LIN {X 0,Y 177.073,Z 822.923,A -85,B 0,C 180,E1 -26070.539,E2 -26070.539} C_VEL
LIN {X 0,Y 180.629,Z 808.52,A -85,B 0,C 180,E1 -26071.33,E2 -26071.33} C_VEL
LIN {X 0,Y 182.9,Z 794.433,A -85,B 0,C 180,E1 -26071.841,E2 -26071.841} C_VEL
LIN {X 0,Y 185.471,Z 767.507,A -85,B 0,C 180,E1 -26072.606,E2 -26072.606} C_VEL
LIN {X 0,Y 182.681,Z 759.244,A -85,B 0,C 180,E1 -26075.344,E2 -26075.344} C_VEL
LIN {X 0,Y 179.682,Z 751.238,A -85,B 0,C 180,E1 -26078.707,E2 -26078.707} C_VEL
LIN {X 0,Y 177.784,Z 746.896,A -85,B 0,C 180,E1 -26081.141,E2 -26081.141} C_VEL
LIN {X 0,Y 176.059,Z 743.86,A -85,B 0,C 180,E1 -26083.611,E2 -26083.611} C_VEL
LIN {X 0,Y 174.842,Z 741.596,A -85,B 0,C 180,E1 -26085.711,E2 -26085.711} C_VEL
LIN {X 0,Y 172.904,Z 737.776,A -85,B 0,C 180,E1 -26090.311,E2 -26090.311} C_VEL
LIN {X 0,Y 171.638,Z 736.041,A -85,B 0,C 180,E1 -26097.654,E2 -26097.654} C_VEL
LIN {X 0,Y 171.809,Z 736.329,A -85,B 0,C 180,E1 -26100.587,E2 -26100.587} C_VEL
LIN {X 0,Y 173.048,Z 737.983,A -85,B 0,C 180,E1 -26105.682,E2 -26105.682} C_VEL
LIN {X 0,Y 174.768,Z 741.458,A -85,B 0,C 180,E1 -26109.725,E2 -26109.725} C_VEL
LIN {X 0,Y 175.622,Z 743.043,A -85,B 0,C 180,E1 -26111.251,E2 -26111.251} C_VEL
LIN {X 0,Y 177.589,Z 746.529,A -85,B 0,C 180,E1 -26114.175,E2 -26114.175} C_VEL
LIN {X 0,Y 180.001,Z 750.965,A -85,B 0,C 180,E1 -26117.129,E2 -26117.129} C_VEL
LIN {X 0,Y 183.401,Z 757.678,A -85,B 0,C 180,E1 -26120.615,E2 -26120.615} C_VEL
LIN {X 0,Y 185.832,Z 763.005,A -85,B 0,C 180,E1 -26122.807,E2 -26122.807} C_VEL
LIN {X 0,Y 182.965,Z 792.297,A -85,B 0,C 180,E1 -26123.684,E2 -26123.684} C_VEL
LIN {X 0,Y 180.308,Z 806.858,A -85,B 0,C 180,E1 -26124.351,E2 -26124.351} C_VEL
LIN {X 0,Y 176.455,Z 821.351,A -85,B 0,C 180,E1 -26125.363,E2 -26125.363} C_VEL
LIN {X 0,Y 171.502,Z 834.975,A -85,B 0,C 180,E1 -26126.6,E2 -26126.6} C_VEL
LIN {X 0,Y 166.318,Z 846.673,A -85,B 0,C 180,E1 -26128.103,E2 -26128.103} C_VEL
LIN {X 0,Y 160.284,Z 858.049,A -85,B 0,C 180,E1 -26130.005,E2 -26130.005} C_VEL
LIN {X 0,Y 153.748,Z 868.482,A -85,B 0,C 180,E1 -26132.258,E2 -26132.258} C_VEL
LIN {X 0,Y 146.256,Z 878.831,A -85,B 0,C 180,E1 -26135.225,E2 -26135.225} C_VEL
LIN {X 0,Y 139.276,Z 887.346,A -85,B 0,C 180,E1 -26138.543,E2 -26138.543} C_VEL
LIN {X 0,Y 131.602,Z 895.448,A -85,B 0,C 180,E1 -26142.752,E2 -26142.752} C_VEL
LIN {X 0,Y 124.73,Z 901.95,A -85,B 0,C 180,E1 -26147.457,E2 -26147.457} C_VEL
LIN {X 0,Y 117.992,Z 907.69,A -85,B 0,C 180,E1 -26153.443,E2 -26153.443} C_VEL
LIN {X 0,Y 112.636,Z 911.844,A -85,B 0,C 180,E1 -26160.055,E2 -26160.055} C_VEL
LIN {X 0,Y 108.658,Z 914.547,A -85,B 0,C 180,E1 -26167.165,E2 -26167.165} C_VEL
LIN {X 0,Y 106.159,Z 915.885,A -85,B 0,C 180,E1 -26174.645,E2 -26174.645} C_VEL
LIN {X 0,Y 105.229,Z 915.893,A -85,B 0,C 180,E1 -26182.324,E2 -26182.324} C_VEL
LIN {X 0,Y 105.422,Z 914.588,A -85,B 0,C 180,E1 -26190,E2 -26190} C_VEL
LIN {X 0,Y 106.561,Z 911.96,A -85,B 0,C 180,E1 -26197.58,E2 -26197.58} C_VEL
LIN {X 0,Y 109.233,Z 907.919,A -85,B 0,C 180,E1 -26204.914,E2 -26204.914} C_VEL
LIN {X 0,Y 112.051,Z 904.063,A -85,B 0,C 180,E1 -26209.989,E2 -26209.989} C_VEL
LIN {X 0,Y 115.769,Z 898.932,A -85,B 0,C 180,E1 -26215.148,E2 -26215.148} C_VEL
LIN {X 0,Y 120.816,Z 891.816,A -85,B 0,C 180,E1 -26220.597,E2 -26220.597} C_VEL
LIN {X 0,Y 127.127,Z 882.991,A -85,B 0,C 180,E1 -26225.485,E2 -26225.485} C_VEL
LIN {X 0,Y 133.06,Z 873.738,A -85,B 0,C 180,E1 -26229.333,E2 -26229.333} C_VEL
LIN {X 0,Y 138.745,Z 863.523,A -85,B 0,C 180,E1 -26232.649,E2 -26232.649} C_VEL
LIN {X 0,Y 142.557,Z 855.85,A -85,B 0,C 180,E1 -26234.63,E2 -26234.63} C_VEL
LIN {X 0,Y 147.858,Z 844.228,A -85,B 0,C 180,E1 -26236.954,E2 -26236.954} C_VEL
LIN {X 0,Y 152.056,Z 833.202,A -85,B 0,C 180,E1 -26238.684,E2 -26238.684} C_VEL
LIN {X 0,Y 156.398,Z 819.272,A -85,B 0,C 180,E1 -26240.313,E2 -26240.313} C_VEL
LIN {X 0,Y 159.627,Z 805.18,A -85,B 0,C 180,E1 -26241.524,E2 -26241.524} C_VEL
LIN {X 0,Y 161.82,Z 791.195,A -85,B 0,C 180,E1 -26242.321,E2 -26242.321} C_VEL
LIN {X 0,Y 165.759,Z 746.595,A -85,B 0,C 180,E1 -26243.808,E2 -26243.808} C_VEL
LIN {X 0,Y 161.599,Z 737.779,A -85,B 0,C 180,E1 -26246.875,E2 -26246.875} C_VEL
LIN {X 0,Y 157.468,Z 730.066,A -85,B 0,C 180,E1 -26250.312,E2 -26250.312} C_VEL
LIN {X 0,Y 153.944,Z 723.905,A -85,B 0,C 180,E1 -26253.732,E2 -26253.732} C_VEL
LIN {X 0,Y 151.674,Z 720.327,A -85,B 0,C 180,E1 -26256.257,E2 -26256.257} C_VEL
LIN {X 0,Y 149.381,Z 716.691,A -85,B 0,C 180,E1 -26259.241,E2 -26259.241} C_VEL
LIN {X 0,Y 147.032,Z 713.071,A -85,B 0,C 180,E1 -26263.011,E2 -26263.011} C_VEL
LIN {X 0,Y 144.407,Z 709.358,A -85,B 0,C 180,E1 -26269.192,E2 -26269.192} C_VEL
LIN {X 0,Y 143.974,Z 707.729,A -85,B 0,C 180,E1 -26271.246,E2 -26271.246} C_VEL
LIN {X 0,Y 143.41,Z 707.23,A -85,B 0,C 180,E1 -26279.999,E2 -26279.999} C_VEL
LIN {X 0,Y 144.182,Z 707.95,A -85,B 0,C 180,E1 -26284.105,E2 -26284.105} C_VEL
LIN {X 0,Y 145.926,Z 711.714,A -85,B 0,C 180,E1 -26289.355,E2 -26289.355} C_VEL
LIN {X 0,Y 147.111,Z 713.082,A -85,B 0,C 180,E1 -26291.617,E2 -26291.617} C_VEL
LIN {X 0,Y 149.448,Z 716.686,A -85,B 0,C 180,E1 -26295.338,E2 -26295.338} C_VEL
LIN {X 0,Y 152.699,Z 721.894,A -85,B 0,C 180,E1 -26299.414,E2 -26299.414} C_VEL
LIN {X 0,Y 156.291,Z 727.806,A -85,B 0,C 180,E1 -26303.082,E2 -26303.082} C_VEL
LIN {X 0,Y 158.506,Z 732.054,A -85,B 0,C 180,E1 -26305.103,E2 -26305.103} C_VEL
LIN {X 0,Y 161.92,Z 740.882,A -85,B 0,C 180,E1 -26308.077,E2 -26308.077} C_VEL
LIN {X 0,Y 165.49,Z 751.393,A -85,B 0,C 180,E1 -26310.914,E2 -26310.914} C_VEL
LIN {X 0,Y 161.322,Z 798.641,A -85,B 0,C 180,E1 -26312.498,E2 -26312.498} C_VEL
LIN {X 0,Y 158.933,Z 812.957,A -85,B 0,C 180,E1 -26313.276,E2 -26313.276} C_VEL
LIN {X 0,Y 155.415,Z 827.05,A -85,B 0,C 180,E1 -26314.382,E2 -26314.382} C_VEL
LIN {X 0,Y 150.891,Z 841.025,A -85,B 0,C 180,E1 -26315.975,E2 -26315.975} C_VEL
LIN {X 0,Y 145.821,Z 853.521,A -85,B 0,C 180,E1 -26317.888,E2 -26317.888} C_VEL
LIN {X 0,Y 140.409,Z 864.953,A -85,B 0,C 180,E1 -26320.241,E2 -26320.241} C_VEL
LIN {X 0,Y 134.823,Z 875.474,A -85,B 0,C 180,E1 -26323.131,E2 -26323.131} C_VEL
LIN {X 0,Y 128.441,Z 885.919,A -85,B 0,C 180,E1 -26326.844,E2 -26326.844} C_VEL
LIN {X 0,Y 122.678,Z 894.538,A -85,B 0,C 180,E1 -26330.937,E2 -26330.937} C_VEL
LIN {X 0,Y 116.942,Z 902.78,A -85,B 0,C 180,E1 -26336.226,E2 -26336.226} C_VEL
LIN {X 0,Y 112.117,Z 909.461,A -85,B 0,C 180,E1 -26342.013,E2 -26342.013} C_VEL
LIN {X 0,Y 108.319,Z 915.314,A -85,B 0,C 180,E1 -26349.092,E2 -26349.092} C_VEL
LIN {X 0,Y 106.388,Z 918.704,A -85,B 0,C 180,E1 -26354.678,E2 -26354.678} C_VEL
LIN {X 0,Y 105.229,Z 921.879,A -85,B 0,C 180,E1 -26362.323,E2 -26362.323} C_VEL
LIN {X 0,Y 105.149,Z 922.938,A -85,B 0,C 180,E1 -26366.167,E2 -26366.167} C_VEL
LIN {X 0,Y 105.301,Z 923.651,A -85,B 0,C 180,E1 -26370,E2 -26370} C_VEL
LIN {X 0,Y 105.224,Z 924.013,A -85,B 0,C 180,E1 -26377.676,E2 -26377.676} C_VEL
LIN {X 0,Y 106.436,Z 923.042,A -85,B 0,C 180,E1 -26385.314,E2 -26385.314} C_VEL
LIN {X 0,Y 109.333,Z 920.744,A -85,B 0,C 180,E1 -26392.686,E2 -26392.686} C_VEL
LIN {X 0,Y 113.857,Z 917.06,A -85,B 0,C 180,E1 -26399.591,E2 -26399.591} C_VEL
LIN {X 0,Y 119.273,Z 912.338,A -85,B 0,C 180,E1 -26405.452,E2 -26405.452} C_VEL
LIN {X 0,Y 121.304,Z 910.059,A -85,B 0,C 180,E1 -26407.862,E2 -26407.862} C_VEL
LIN {X 0,Y 123.493,Z 906.012,A -85,B 0,C 180,E1 -26411.974,E2 -26411.974} C_VEL
LIN {X 0,Y 126.146,Z 901.426,A -85,B 0,C 180,E1 -26415.814,E2 -26415.814} C_VEL
LIN {X 0,Y 128.79,Z 898.306,A -85,B 0,C 180,E1 -26417.725,E2 -26417.725} C_VEL
LIN {X 0,Y 136.909,Z 889.585,A -85,B 0,C 180,E1 -26421.521,E2 -26421.521} C_VEL
LIN {X 0,Y 144.395,Z 880.343,A -85,B 0,C 180,E1 -26424.492,E2 -26424.492} C_VEL
LIN {X 0,Y 151.862,Z 869.757,A -85,B 0,C 180,E1 -26427.014,E2 -26427.014} C_VEL
LIN {X 0,Y 158.865,Z 858.295,A -85,B 0,C 180,E1 -26428.995,E2 -26428.995} C_VEL
LIN {X 0,Y 164.572,Z 847.189,A -85,B 0,C 180,E1 -26430.471,E2 -26430.471} C_VEL
LIN {X 0,Y 169.642,Z 835.263,A -85,B 0,C 180,E1 -26431.685,E2 -26431.685} C_VEL
LIN {X 0,Y 174.075,Z 822.227,A -85,B 0,C 180,E1 -26432.65,E2 -26432.65} C_VEL
LIN {X 0,Y 177.7,Z 807.753,A -85,B 0,C 180,E1 -26433.406,E2 -26433.406} C_VEL
LIN {X 0,Y 179.983,Z 793.525,A -85,B 0,C 180,E1 -26433.91,E2 -26433.91} C_VEL
LIN {X 0,Y 182.27,Z 770.597,A -85,B 0,C 180,E1 -26434.526,E2 -26434.526} C_VEL
LIN {X 0,Y 179.677,Z 762.653,A -85,B 0,C 180,E1 -26437.393,E2 -26437.393} C_VEL
LIN {X 0,Y 177.483,Z 756.512,A -85,B 0,C 180,E1 -26440.166,E2 -26440.166} C_VEL
LIN {X 0,Y 176.003,Z 752.899,A -85,B 0,C 180,E1 -26442.274,E2 -26442.274} C_VEL
LIN {X 0,Y 173.64,Z 748.379,A -85,B 0,C 180,E1 -26446.261,E2 -26446.261} C_VEL
LIN {X 0,Y 171.931,Z 744.757,A -85,B 0,C 180,E1 -26450.59,E2 -26450.59} C_VEL
LIN {X 0,Y 170.77,Z 743.1,A -85,B 0,C 180,E1 -26457.642,E2 -26457.642} C_VEL
LIN {X 0,Y 170.939,Z 743.403,A -85,B 0,C 180,E1 -26460.59,E2 -26460.59} C_VEL
LIN {X 0,Y 171.974,Z 744.847,A -85,B 0,C 180,E1 -26465.13,E2 -26465.13} C_VEL
LIN {X 0,Y 173.727,Z 748.455,A -85,B 0,C 180,E1 -26469.47,E2 -26469.47} C_VEL
LIN {X 0,Y 176.152,Z 753.196,A -85,B 0,C 180,E1 -26473.52,E2 -26473.52} C_VEL
LIN {X 0,Y 178.871,Z 758.486,A -85,B 0,C 180,E1 -26476.992,E2 -26476.992} C_VEL
LIN {X 0,Y 182.507,Z 766.355,A -85,B 0,C 180,E1 -26480.809,E2 -26480.809} C_VEL
LIN {X 0,Y 182.607,Z 766.645,A -85,B 0,C 180,E1 -26480.911,E2 -26480.911} C_VEL
LIN {X 0,Y 179.863,Z 793.134,A -85,B 0,C 180,E1 -26481.688,E2 -26481.688} C_VEL
LIN {X 0,Y 177.112,Z 807.587,A -85,B 0,C 180,E1 -26482.34,E2 -26482.34} C_VEL
LIN {X 0,Y 173.154,Z 821.94,A -85,B 0,C 180,E1 -26483.321,E2 -26483.321} C_VEL
LIN {X 0,Y 168.297,Z 834.919,A -85,B 0,C 180,E1 -26484.459,E2 -26484.459} C_VEL
LIN {X 0,Y 163.066,Z 846.428,A -85,B 0,C 180,E1 -26485.882,E2 -26485.882} C_VEL
LIN {X 0,Y 156.137,Z 859.073,A -85,B 0,C 180,E1 -26487.95,E2 -26487.95} C_VEL
LIN {X 0,Y 150.035,Z 868.401,A -85,B 0,C 180,E1 -26489.936,E2 -26489.936} C_VEL
LIN {X 0,Y 142.248,Z 878.818,A -85,B 0,C 180,E1 -26492.869,E2 -26492.869} C_VEL
LIN {X 0,Y 134.919,Z 887.383,A -85,B 0,C 180,E1 -26496.158,E2 -26496.158} C_VEL
LIN {X 0,Y 126.828,Z 895.54,A -85,B 0,C 180,E1 -26500.365,E2 -26500.365} C_VEL
LIN {X 0,Y 119.532,Z 902.079,A -85,B 0,C 180,E1 -26505.126,E2 -26505.126} C_VEL
LIN {X 0,Y 112.286,Z 907.853,A -85,B 0,C 180,E1 -26511.252,E2 -26511.252} C_VEL
LIN {X 0,Y 106.461,Z 912.039,A -85,B 0,C 180,E1 -26518.122,E2 -26518.122} C_VEL
LIN {X 0,Y 102.067,Z 914.772,A -85,B 0,C 180,E1 -26525.598,E2 -26525.598} C_VEL
LIN {X 0,Y 99.251,Z 916.139,A -85,B 0,C 180,E1 -26533.547,E2 -26533.547} C_VEL
LIN {X 0,Y 98.161,Z 916.177,A -85,B 0,C 180,E1 -26541.768,E2 -26541.768} C_VEL
LIN {X 0,Y 98.316,Z 914.907,A -85,B 0,C 180,E1 -26550,E2 -26550} C_VEL
LIN {X 0,Y 99.549,Z 912.313,A -85,B 0,C 180,E1 -26558.118,E2 -26558.118} C_VEL
LIN {X 0,Y 102.417,Z 908.303,A -85,B 0,C 180,E1 -26565.932,E2 -26565.932} C_VEL
LIN {X 0,Y 105.534,Z 904.324,A -85,B 0,C 180,E1 -26571.486,E2 -26571.486} C_VEL
LIN {X 0,Y 109.397,Z 899.368,A -85,B 0,C 180,E1 -26576.725,E2 -26576.725} C_VEL
LIN {X 0,Y 114.789,Z 892.289,A -85,B 0,C 180,E1 -26582.393,E2 -26582.393} C_VEL
LIN {X 0,Y 121.449,Z 883.509,A -85,B 0,C 180,E1 -26587.418,E2 -26587.418} C_VEL
LIN {X 0,Y 127.682,Z 874.314,A -85,B 0,C 180,E1 -26591.34,E2 -26591.34} C_VEL
LIN {X 0,Y 133.645,Z 864.172,A -85,B 0,C 180,E1 -26594.697,E2 -26594.697} C_VEL
LIN {X 0,Y 137.63,Z 856.543,A -85,B 0,C 180,E1 -26596.692,E2 -26596.692} C_VEL
LIN {X 0,Y 143.12,Z 845.016,A -85,B 0,C 180,E1 -26599.026,E2 -26599.026} C_VEL
LIN {X 0,Y 148.149,Z 832.352,A -85,B 0,C 180,E1 -26600.97,E2 -26600.97} C_VEL
LIN {X 0,Y 152.321,Z 819.233,A -85,B 0,C 180,E1 -26602.469,E2 -26602.469} C_VEL
LIN {X 0,Y 155.676,Z 805.031,A -85,B 0,C 180,E1 -26603.665,E2 -26603.665} C_VEL
LIN {X 0,Y 157.936,Z 790.7,A -85,B 0,C 180,E1 -26604.46,E2 -26604.46} C_VEL
LIN {X 0,Y 161.683,Z 750.383,A -85,B 0,C 180,E1 -26605.753,E2 -26605.753} C_VEL
LIN {X 0,Y 161.578,Z 749.318,A -85,B 0,C 180,E1 -26605.904,E2 -26605.904} C_VEL
LIN {X 0,Y 157.893,Z 741.409,A -85,B 0,C 180,E1 -26608.92,E2 -26608.92} C_VEL
LIN {X 0,Y 153.683,Z 733.209,A -85,B 0,C 180,E1 -26612.898,E2 -26612.898} C_VEL
LIN {X 0,Y 150.227,Z 727.144,A -85,B 0,C 180,E1 -26616.813,E2 -26616.813} C_VEL
LIN {X 0,Y 147.749,Z 723.204,A -85,B 0,C 180,E1 -26620.212,E2 -26620.212} C_VEL
LIN {X 0,Y 145.313,Z 719.255,A -85,B 0,C 180,E1 -26624.549,E2 -26624.549} C_VEL
LIN {X 0,Y 143.413,Z 716.402,A -85,B 0,C 180,E1 -26629.537,E2 -26629.537} C_VEL
LIN {X 0,Y 143.022,Z 714.868,A -85,B 0,C 180,E1 -26631.522,E2 -26631.522} C_VEL
LIN {X 0,Y 142.542,Z 714.285,A -85,B 0,C 180,E1 -26639.999,E2 -26639.999} C_VEL
LIN {X 0,Y 143.167,Z 714.938,A -85,B 0,C 180,E1 -26643.583,E2 -26643.583} C_VEL
LIN {X 0,Y 144.958,Z 718.789,A -85,B 0,C 180,E1 -26649.207,E2 -26649.207} C_VEL
LIN {X 0,Y 145.799,Z 719.875,A -85,B 0,C 180,E1 -26650.906,E2 -26650.906} C_VEL
LIN {X 0,Y 148.461,Z 724.292,A -85,B 0,C 180,E1 -26655.333,E2 -26655.333} C_VEL
LIN {X 0,Y 151.218,Z 728.929,A -85,B 0,C 180,E1 -26658.897,E2 -26658.897} C_VEL
LIN {X 0,Y 154.178,Z 734.124,A -85,B 0,C 180,E1 -26662.1,E2 -26662.1} C_VEL
LIN {X 0,Y 156.02,Z 737.94,A -85,B 0,C 180,E1 -26663.916,E2 -26663.916} C_VEL
LIN {X 0,Y 159.188,Z 746.807,A -85,B 0,C 180,E1 -26666.916,E2 -26666.916} C_VEL
LIN {X 0,Y 161.451,Z 753.905,A -85,B 0,C 180,E1 -26668.899,E2 -26668.899} C_VEL
LIN {X 0,Y 157.348,Z 798.562,A -85,B 0,C 180,E1 -26670.39,E2 -26670.39} C_VEL
LIN {X 0,Y 154.79,Z 813.184,A -85,B 0,C 180,E1 -26671.176,E2 -26671.176} C_VEL
LIN {X 0,Y 151.159,Z 827.148,A -85,B 0,C 180,E1 -26672.262,E2 -26672.262} C_VEL
LIN {X 0,Y 146.8,Z 840.151,A -85,B 0,C 180,E1 -26673.713,E2 -26673.713} C_VEL
LIN {X 0,Y 141.543,Z 852.763,A -85,B 0,C 180,E1 -26675.603,E2 -26675.603} C_VEL
LIN {X 0,Y 135.899,Z 864.281,A -85,B 0,C 180,E1 -26677.94,E2 -26677.94} C_VEL
LIN {X 0,Y 130.037,Z 874.868,A -85,B 0,C 180,E1 -26680.83,E2 -26680.83} C_VEL
LIN {X 0,Y 123.323,Z 885.374,A -85,B 0,C 180,E1 -26684.572,E2 -26684.572} C_VEL
LIN {X 0,Y 117.181,Z 894.037,A -85,B 0,C 180,E1 -26688.72,E2 -26688.72} C_VEL
LIN {X 0,Y 111.064,Z 902.336,A -85,B 0,C 180,E1 -26694.173,E2 -26694.173} C_VEL
LIN {X 0,Y 105.664,Z 909.265,A -85,B 0,C 180,E1 -26700.426,E2 -26700.426} C_VEL
LIN {X 0,Y 101.675,Z 914.936,A -85,B 0,C 180,E1 -26707.655,E2 -26707.655} C_VEL
LIN {X 0,Y 99.504,Z 918.354,A -85,B 0,C 180,E1 -26713.589,E2 -26713.589} C_VEL
LIN {X 0,Y 98.171,Z 921.558,A -85,B 0,C 180,E1 -26721.768,E2 -26721.768} C_VEL
LIN {X 0,Y 98.066,Z 922.632,A -85,B 0,C 180,E1 -26725.89,E2 -26725.89} C_VEL
LIN {X 0,Y 98.2,Z 923.358,A -85,B 0,C 180,E1 -26730,E2 -26730} C_VEL
LIN {X 0,Y 98.167,Z 923.745,A -85,B 0,C 180,E1 -26738.232,E2 -26738.232} C_VEL
LIN {X 0,Y 99.572,Z 922.801,A -85,B 0,C 180,E1 -26746.399,E2 -26746.399} C_VEL
LIN {X 0,Y 102.778,Z 920.529,A -85,B 0,C 180,E1 -26754.222,E2 -26754.222} C_VEL
LIN {X 0,Y 107.673,Z 916.874,A -85,B 0,C 180,E1 -26761.478,E2 -26761.478} C_VEL
LIN {X 0,Y 114.069,Z 911.733,A -85,B 0,C 180,E1 -26768.033,E2 -26768.033} C_VEL
LIN {X 0,Y 119.82,Z 906.784,A -85,B 0,C 180,E1 -26772.417,E2 -26772.417} C_VEL
LIN {X 0,Y 127.356,Z 899.704,A -85,B 0,C 180,E1 -26776.986,E2 -26776.986} C_VEL
LIN {X 0,Y 128.79,Z 898.306,A -85,B 0,C 180,E1 -26777.725,E2 -26777.725} C_VEL
LIN {X 0,Y 131.53,Z 895.029,A -85,B 0,C 180,E1 -26779.529,E2 -26779.529} C_VEL
LIN {X 0,Y 134.869,Z 889.483,A -85,B 0,C 180,E1 -26782.77,E2 -26782.77} C_VEL
LIN {X 0,Y 138.31,Z 883.455,A -85,B 0,C 180,E1 -26785.745,E2 -26785.745} C_VEL
LIN {X 0,Y 141.092,Z 879.427,A -85,B 0,C 180,E1 -26787.104,E2 -26787.104} C_VEL
LIN {X 0,Y 148.829,Z 868.775,A -85,B 0,C 180,E1 -26789.519,E2 -26789.519} C_VEL
LIN {X 0,Y 156.04,Z 857.167,A -85,B 0,C 180,E1 -26791.435,E2 -26791.435} C_VEL
LIN {X 0,Y 162.684,Z 844.289,A -85,B 0,C 180,E1 -26793,E2 -26793} C_VEL
LIN {X 0,Y 168.302,Z 830.696,A -85,B 0,C 180,E1 -26794.212,E2 -26794.212} C_VEL
LIN {X 0,Y 172.636,Z 817.104,A -85,B 0,C 180,E1 -26795.067,E2 -26795.067} C_VEL
LIN {X 0,Y 175.903,Z 802.401,A -85,B 0,C 180,E1 -26795.724,E2 -26795.724} C_VEL
LIN {X 0,Y 177.927,Z 787.042,A -85,B 0,C 180,E1 -26796.179,E2 -26796.179} C_VEL
LIN {X 0,Y 179.248,Z 773.696,A -85,B 0,C 180,E1 -26796.538,E2 -26796.538} C_VEL
LIN {X 0,Y 176.676,Z 765.423,A -85,B 0,C 180,E1 -26799.821,E2 -26799.821} C_VEL
LIN {X 0,Y 174.789,Z 760.013,A -85,B 0,C 180,E1 -26802.638,E2 -26802.638} C_VEL
LIN {X 0,Y 172.66,Z 755.489,A -85,B 0,C 180,E1 -26806.405,E2 -26806.405} C_VEL
LIN {X 0,Y 170.88,Z 751.655,A -85,B 0,C 180,E1 -26811.128,E2 -26811.128} C_VEL
LIN {X 0,Y 169.903,Z 750.158,A -85,B 0,C 180,E1 -26817.63,E2 -26817.63} C_VEL
LIN {X 0,Y 170.103,Z 750.573,A -85,B 0,C 180,E1 -26820.888,E2 -26820.888} C_VEL
LIN {X 0,Y 170.992,Z 751.965,A -85,B 0,C 180,E1 -26824.864,E2 -26824.864} C_VEL
LIN {X 0,Y 172.819,Z 755.943,A -85,B 0,C 180,E1 -26829.52,E2 -26829.52} C_VEL
LIN {X 0,Y 174.701,Z 759.82,A -85,B 0,C 180,E1 -26832.802,E2 -26832.802} C_VEL
LIN {X 0,Y 177.124,Z 764.87,A -85,B 0,C 180,E1 -26836.127,E2 -26836.127} C_VEL
LIN {X 0,Y 179.522,Z 770.357,A -85,B 0,C 180,E1 -26838.902,E2 -26838.902} C_VEL
LIN {X 0,Y 177.057,Z 793.466,A -85,B 0,C 180,E1 -26839.598,E2 -26839.598} C_VEL
LIN {X 0,Y 174.237,Z 807.881,A -85,B 0,C 180,E1 -26840.225,E2 -26840.225} C_VEL
LIN {X 0,Y 170.45,Z 821.39,A -85,B 0,C 180,E1 -26841.113,E2 -26841.113} C_VEL
LIN {X 0,Y 165.339,Z 834.849,A -85,B 0,C 180,E1 -26842.233,E2 -26842.233} C_VEL
LIN {X 0,Y 160.067,Z 846.182,A -85,B 0,C 180,E1 -26843.574,E2 -26843.574} C_VEL
LIN {X 0,Y 153.615,Z 857.742,A -85,B 0,C 180,E1 -26845.368,E2 -26845.368} C_VEL
LIN {X 0,Y 146.585,Z 868.32,A -85,B 0,C 180,E1 -26847.504,E2 -26847.504} C_VEL
LIN {X 0,Y 138.484,Z 878.798,A -85,B 0,C 180,E1 -26850.374,E2 -26850.374} C_VEL
LIN {X 0,Y 130.81,Z 887.413,A -85,B 0,C 180,E1 -26853.617,E2 -26853.617} C_VEL
LIN {X 0,Y 122.3,Z 895.633,A -85,B 0,C 180,E1 -26857.801,E2 -26857.801} C_VEL
LIN {X 0,Y 114.546,Z 902.208,A -85,B 0,C 180,E1 -26862.586,E2 -26862.586} C_VEL
LIN {X 0,Y 106.76,Z 908.016,A -85,B 0,C 180,E1 -26868.83,E2 -26868.83} C_VEL
LIN {X 0,Y 100.404,Z 912.235,A -85,B 0,C 180,E1 -26875.946,E2 -26875.946} C_VEL
LIN {X 0,Y 95.565,Z 914.998,A -85,B 0,C 180,E1 -26883.817,E2 -26883.817} C_VEL
LIN {X 0,Y 92.389,Z 916.393,A -85,B 0,C 180,E1 -26892.286,E2 -26892.286} C_VEL
LIN {X 0,Y 91.101,Z 916.458,A -85,B 0,C 180,E1 -26901.125,E2 -26901.125} C_VEL
LIN {X 0,Y 91.219,Z 915.221,A -85,B 0,C 180,E1 -26910,E2 -26910} C_VEL
LIN {X 0,Y 92.549,Z 912.664,A -85,B 0,C 180,E1 -26918.736,E2 -26918.736} C_VEL
LIN {X 0,Y 95.632,Z 908.687,A -85,B 0,C 180,E1 -26927.096,E2 -26927.096} C_VEL
LIN {X 0,Y 98.977,Z 904.725,A -85,B 0,C 180,E1 -26932.988,E2 -26932.988} C_VEL
LIN {X 0,Y 103.132,Z 899.803,A -85,B 0,C 180,E1 -26938.491,E2 -26938.491} C_VEL
LIN {X 0,Y 108.891,Z 892.761,A -85,B 0,C 180,E1 -26944.385,E2 -26944.385} C_VEL
LIN {X 0,Y 115.923,Z 884.023,A -85,B 0,C 180,E1 -26949.538,E2 -26949.538} C_VEL
LIN {X 0,Y 122.476,Z 874.88,A -85,B 0,C 180,E1 -26953.519,E2 -26953.519} C_VEL
LIN {X 0,Y 128.731,Z 864.807,A -85,B 0,C 180,E1 -26956.904,E2 -26956.904} C_VEL
LIN {X 0,Y 132.895,Z 857.235,A -85,B 0,C 180,E1 -26958.903,E2 -26958.903} C_VEL
LIN {X 0,Y 138.589,Z 845.801,A -85,B 0,C 180,E1 -26961.232,E2 -26961.232} C_VEL
LIN {X 0,Y 143.816,Z 833.258,A -85,B 0,C 180,E1 -26963.151,E2 -26963.151} C_VEL
LIN {X 0,Y 148.138,Z 820.316,A -85,B 0,C 180,E1 -26964.629,E2 -26964.629} C_VEL
LIN {X 0,Y 151.613,Z 806.399,A -85,B 0,C 180,E1 -26965.807,E2 -26965.807} C_VEL
LIN {X 0,Y 154.074,Z 792.037,A -85,B 0,C 180,E1 -26966.617,E2 -26966.617} C_VEL
LIN {X 0,Y 157.813,Z 752.619,A -85,B 0,C 180,E1 -26967.932,E2 -26967.932} C_VEL
LIN {X 0,Y 154.16,Z 744.623,A -85,B 0,C 180,E1 -26971.285,E2 -26971.285} C_VEL
LIN {X 0,Y 150.312,Z 736.877,A -85,B 0,C 180,E1 -26975.458,E2 -26975.458} C_VEL
LIN {X 0,Y 147.838,Z 732.613,A -85,B 0,C 180,E1 -26978.637,E2 -26978.637} C_VEL
LIN {X 0,Y 146.181,Z 729.715,A -85,B 0,C 180,E1 -26981.176,E2 -26981.176} C_VEL
LIN {X 0,Y 144.101,Z 726.071,A -85,B 0,C 180,E1 -26985.191,E2 -26985.191} C_VEL
LIN {X 0,Y 142.332,Z 723.152,A -85,B 0,C 180,E1 -26990.303,E2 -26990.303} C_VEL
LIN {X 0,Y 142.03,Z 721.788,A -85,B 0,C 180,E1 -26992.106,E2 -26992.106} C_VEL
LIN {X 0,Y 141.678,Z 721.311,A -85,B 0,C 180,E1 -26999.999,E2 -26999.999} C_VEL
LIN {X 0,Y 142.17,Z 721.881,A -85,B 0,C 180,E1 -27003.054,E2 -27003.054} C_VEL
LIN {X 0,Y 143.805,Z 725.652,A -85,B 0,C 180,E1 -27008.643,E2 -27008.643} C_VEL
LIN {X 0,Y 144.592,Z 726.849,A -85,B 0,C 180,E1 -27010.364,E2 -27010.364} C_VEL
LIN {X 0,Y 146.858,Z 730.79,A -85,B 0,C 180,E1 -27014.395,E2 -27014.395} C_VEL
LIN {X 0,Y 149.399,Z 735.345,A -85,B 0,C 180,E1 -27017.937,E2 -27017.937} C_VEL
LIN {X 0,Y 152.045,Z 740.252,A -85,B 0,C 180,E1 -27021.013,E2 -27021.013} C_VEL
LIN {X 0,Y 153.558,Z 743.659,A -85,B 0,C 180,E1 -27022.638,E2 -27022.638} C_VEL
LIN {X 0,Y 156.452,Z 752.491,A -85,B 0,C 180,E1 -27025.644,E2 -27025.644} C_VEL
LIN {X 0,Y 157.605,Z 756.445,A -85,B 0,C 180,E1 -27026.775,E2 -27026.775} C_VEL
LIN {X 0,Y 153.57,Z 798.621,A -85,B 0,C 180,E1 -27028.178,E2 -27028.178} C_VEL
LIN {X 0,Y 151.047,Z 812.646,A -85,B 0,C 180,E1 -27028.917,E2 -27028.917} C_VEL
LIN {X 0,Y 147.47,Z 826.108,A -85,B 0,C 180,E1 -27029.914,E2 -27029.914} C_VEL
LIN {X 0,Y 142.958,Z 839.278,A -85,B 0,C 180,E1 -27031.33,E2 -27031.33} C_VEL
LIN {X 0,Y 137.52,Z 852.008,A -85,B 0,C 180,E1 -27033.19,E2 -27033.19} C_VEL
LIN {X 0,Y 131.608,Z 863.606,A -85,B 0,C 180,E1 -27035.475,E2 -27035.475} C_VEL
LIN {X 0,Y 125.468,Z 874.262,A -85,B 0,C 180,E1 -27038.353,E2 -27038.353} C_VEL
LIN {X 0,Y 118.418,Z 884.824,A -85,B 0,C 180,E1 -27042.109,E2 -27042.109} C_VEL
LIN {X 0,Y 111.883,Z 893.531,A -85,B 0,C 180,E1 -27046.292,E2 -27046.292} C_VEL
LIN {X 0,Y 105.353,Z 901.89,A -85,B 0,C 180,E1 -27051.898,E2 -27051.898} C_VEL
LIN {X 0,Y 99.7,Z 908.543,A -85,B 0,C 180,E1 -27058.018,E2 -27058.018} C_VEL
LIN {X 0,Y 96.082,Z 913.232,A -85,B 0,C 180,E1 -27063.967,E2 -27063.967} C_VEL
LIN {X 0,Y 92.666,Z 917.998,A -85,B 0,C 180,E1 -27072.34,E2 -27072.34} C_VEL
LIN {X 0,Y 91.119,Z 921.237,A -85,B 0,C 180,E1 -27081.126,E2 -27081.126} C_VEL
LIN {X 0,Y 90.98,Z 922.325,A -85,B 0,C 180,E1 -27085.569,E2 -27085.569} C_VEL
LIN {X 0,Y 91.111,Z 923.065,A -85,B 0,C 180,E1 -27090,E2 -27090} C_VEL
LIN {X 0,Y 91.117,Z 923.477,A -85,B 0,C 180,E1 -27098.874,E2 -27098.874} C_VEL
LIN {X 0,Y 92.736,Z 922.56,A -85,B 0,C 180,E1 -27107.646,E2 -27107.646} C_VEL
LIN {X 0,Y 96.312,Z 920.316,A -85,B 0,C 180,E1 -27115.965,E2 -27115.965} C_VEL
LIN {X 0,Y 101.625,Z 916.688,A -85,B 0,C 180,E1 -27123.59,E2 -27123.59} C_VEL
LIN {X 0,Y 108.52,Z 911.578,A -85,B 0,C 180,E1 -27130.362,E2 -27130.362} C_VEL
LIN {X 0,Y 116.8,Z 904.836,A -85,B 0,C 180,E1 -27136.224,E2 -27136.224} C_VEL
LIN {X 0,Y 125.043,Z 897.346,A -85,B 0,C 180,E1 -27140.607,E2 -27140.607} C_VEL
LIN {X 0,Y 133.798,Z 888.22,A -85,B 0,C 180,E1 -27144.379,E2 -27144.379} C_VEL
LIN {X 0,Y 141.092,Z 879.427,A -85,B 0,C 180,E1 -27147.104,E2 -27147.104} C_VEL
LIN {X 0,Y 143.885,Z 875.298,A -85,B 0,C 180,E1 -27148.378,E2 -27148.378} C_VEL
LIN {X 0,Y 147.364,Z 868.35,A -85,B 0,C 180,E1 -27150.806,E2 -27150.806} C_VEL
LIN {X 0,Y 150.809,Z 861.081,A -85,B 0,C 180,E1 -27153.007,E2 -27153.007} C_VEL
LIN {X 0,Y 153.374,Z 856.309,A -85,B 0,C 180,E1 -27153.904,E2 -27153.904} C_VEL
LIN {X 0,Y 159.597,Z 844.547,A -85,B 0,C 180,E1 -27155.263,E2 -27155.263} C_VEL
LIN {X 0,Y 164.958,Z 832.082,A -85,B 0,C 180,E1 -27156.348,E2 -27156.348} C_VEL
LIN {X 0,Y 169.29,Z 819.323,A -85,B 0,C 180,E1 -27157.15,E2 -27157.15} C_VEL
LIN {X 0,Y 172.819,Z 805.081,A -85,B 0,C 180,E1 -27157.796,E2 -27157.796} C_VEL
LIN {X 0,Y 174.985,Z 791.244,A -85,B 0,C 180,E1 -27158.218,E2 -27158.218} C_VEL
LIN {X 0,Y 176.429,Z 776.975,A -85,B 0,C 180,E1 -27158.619,E2 -27158.619} C_VEL
LIN {X 0,Y 174.164,Z 769.113,A -85,B 0,C 180,E1 -27162.005,E2 -27162.005} C_VEL
LIN {X 0,Y 172.861,Z 765.424,A -85,B 0,C 180,E1 -27164.234,E2 -27164.234} C_VEL
LIN {X 0,Y 171.138,Z 761.753,A -85,B 0,C 180,E1 -27167.701,E2 -27167.701} C_VEL
LIN {X 0,Y 169.896,Z 758.62,A -85,B 0,C 180,E1 -27171.49,E2 -27171.49} C_VEL
LIN {X 0,Y 169.036,Z 757.217,A -85,B 0,C 180,E1 -27177.618,E2 -27177.618} C_VEL
LIN {X 0,Y 169.23,Z 757.677,A -85,B 0,C 180,E1 -27180.893,E2 -27180.893} C_VEL
LIN {X 0,Y 169.98,Z 758.925,A -85,B 0,C 180,E1 -27184.447,E2 -27184.447} C_VEL
LIN {X 0,Y 171.643,Z 762.832,A -85,B 0,C 180,E1 -27189.009,E2 -27189.009} C_VEL
LIN {X 0,Y 173.323,Z 766.532,A -85,B 0,C 180,E1 -27192.143,E2 -27192.143} C_VEL
LIN {X 0,Y 175.535,Z 771.459,A -85,B 0,C 180,E1 -27195.392,E2 -27195.392} C_VEL
LIN {X 0,Y 176.671,Z 774.478,A -85,B 0,C 180,E1 -27196.881,E2 -27196.881} C_VEL
LIN {X 0,Y 174.358,Z 794.644,A -85,B 0,C 180,E1 -27197.477,E2 -27197.477} C_VEL
LIN {X 0,Y 171.347,Z 809.215,A -85,B 0,C 180,E1 -27198.095,E2 -27198.095} C_VEL
LIN {X 0,Y 167.245,Z 823.116,A -85,B 0,C 180,E1 -27199.004,E2 -27199.004} C_VEL
LIN {X 0,Y 162.638,Z 834.784,A -85,B 0,C 180,E1 -27199.932,E2 -27199.932} C_VEL
LIN {X 0,Y 157.337,Z 845.937,A -85,B 0,C 180,E1 -27201.18,E2 -27201.18} C_VEL
LIN {X 0,Y 150.689,Z 857.589,A -85,B 0,C 180,E1 -27202.909,E2 -27202.909} C_VEL
LIN {X 0,Y 143.41,Z 868.24,A -85,B 0,C 180,E1 -27204.959,E2 -27204.959} C_VEL
LIN {X 0,Y 134.992,Z 878.776,A -85,B 0,C 180,E1 -27207.741,E2 -27207.741} C_VEL
LIN {X 0,Y 126.963,Z 887.442,A -85,B 0,C 180,E1 -27210.908,E2 -27210.908} C_VEL
LIN {X 0,Y 118.037,Z 895.722,A -85,B 0,C 180,E1 -27215.047,E2 -27215.047} C_VEL
LIN {X 0,Y 109.826,Z 902.337,A -85,B 0,C 180,E1 -27219.834,E2 -27219.834} C_VEL
LIN {X 0,Y 101.445,Z 908.18,A -85,B 0,C 180,E1 -27226.149,E2 -27226.149} C_VEL
LIN {X 0,Y 94.522,Z 912.43,A -85,B 0,C 180,E1 -27233.5,E2 -27233.5} C_VEL
LIN {X 0,Y 89.169,Z 915.223,A -85,B 0,C 180,E1 -27241.778,E2 -27241.778} C_VEL
LIN {X 0,Y 85.583,Z 916.648,A -85,B 0,C 180,E1 -27250.824,E2 -27250.824} C_VEL
LIN {X 0,Y 84.042,Z 916.741,A -85,B 0,C 180,E1 -27260.372,E2 -27260.372} C_VEL
LIN {X 0,Y 83.902,Z 916.298,A -85,B 0,C 180,E1 -27265.195,E2 -27265.195} C_VEL
LIN {X 0,Y 84.67,Z 914.439,A -85,B 0,C 180,E1 -27274.762,E2 -27274.762} C_VEL
LIN {X 0,Y 86.979,Z 911.227,A -85,B 0,C 180,E1 -27284.029,E2 -27284.029} C_VEL
LIN {X 0,Y 91.286,Z 906.53,A -85,B 0,C 180,E1 -27292.641,E2 -27292.641} C_VEL
LIN {X 0,Y 96.963,Z 900.238,A -85,B 0,C 180,E1 -27300.489,E2 -27300.489} C_VEL
LIN {X 0,Y 103.142,Z 893.233,A -85,B 0,C 180,E1 -27306.6,E2 -27306.6} C_VEL
LIN {X 0,Y 110.572,Z 884.538,A -85,B 0,C 180,E1 -27311.866,E2 -27311.866} C_VEL
LIN {X 0,Y 117.464,Z 875.444,A -85,B 0,C 180,E1 -27315.888,E2 -27315.888} C_VEL
LIN {X 0,Y 124.653,Z 864.427,A -85,B 0,C 180,E1 -27319.565,E2 -27319.565} C_VEL
LIN {X 0,Y 130.956,Z 853.183,A -85,B 0,C 180,E1 -27322.335,E2 -27322.335} C_VEL
LIN {X 0,Y 136.968,Z 840.724,A -85,B 0,C 180,E1 -27324.545,E2 -27324.545} C_VEL
LIN {X 0,Y 141.773,Z 828.674,A -85,B 0,C 180,E1 -27326.134,E2 -27326.134} C_VEL
LIN {X 0,Y 145.883,Z 815.441,A -85,B 0,C 180,E1 -27327.467,E2 -27327.467} C_VEL
LIN {X 0,Y 149.123,Z 801.179,A -85,B 0,C 180,E1 -27328.483,E2 -27328.483} C_VEL
LIN {X 0,Y 151.186,Z 787.067,A -85,B 0,C 180,E1 -27329.127,E2 -27329.127} C_VEL
LIN {X 0,Y 154.148,Z 755.819,A -85,B 0,C 180,E1 -27330.145,E2 -27330.145} C_VEL
LIN {X 0,Y 150.74,Z 748.082,A -85,B 0,C 180,E1 -27333.701,E2 -27333.701} C_VEL
LIN {X 0,Y 147.767,Z 741.984,A -85,B 0,C 180,E1 -27337.357,E2 -27337.357} C_VEL
LIN {X 0,Y 145.076,Z 736.801,A -85,B 0,C 180,E1 -27341.451,E2 -27341.451} C_VEL
LIN {X 0,Y 142.938,Z 732.936,A -85,B 0,C 180,E1 -27345.768,E2 -27345.768} C_VEL
LIN {X 0,Y 141.279,Z 729.912,A -85,B 0,C 180,E1 -27351.069,E2 -27351.069} C_VEL
LIN {X 0,Y 141.02,Z 728.751,A -85,B 0,C 180,E1 -27352.841,E2 -27352.841} C_VEL
LIN {X 0,Y 140.897,Z 728.464,A -85,B 0,C 180,E1 -27360.741,E2 -27360.741} C_VEL
LIN {X 0,Y 141.208,Z 728.944,A -85,B 0,C 180,E1 -27362.68,E2 -27362.68} C_VEL
LIN {X 0,Y 142.77,Z 732.614,A -85,B 0,C 180,E1 -27368.313,E2 -27368.313} C_VEL
LIN {X 0,Y 143.613,Z 734.289,A -85,B 0,C 180,E1 -27370.292,E2 -27370.292} C_VEL
LIN {X 0,Y 145.422,Z 737.52,A -85,B 0,C 180,E1 -27373.648,E2 -27373.648} C_VEL
LIN {X 0,Y 147.841,Z 742.129,A -85,B 0,C 180,E1 -27377.239,E2 -27377.239} C_VEL
LIN {X 0,Y 150.616,Z 747.751,A -85,B 0,C 180,E1 -27380.644,E2 -27380.644} C_VEL
LIN {X 0,Y 153.043,Z 755.603,A -85,B 0,C 180,E1 -27383.502,E2 -27383.502} C_VEL
LIN {X 0,Y 153.99,Z 758.99,A -85,B 0,C 180,E1 -27384.551,E2 -27384.551} C_VEL
LIN {X 0,Y 150.26,Z 797.176,A -85,B 0,C 180,E1 -27385.797,E2 -27385.797} C_VEL
LIN {X 0,Y 147.718,Z 811.335,A -85,B 0,C 180,E1 -27386.485,E2 -27386.485} C_VEL
LIN {X 0,Y 144.046,Z 825.069,A -85,B 0,C 180,E1 -27387.455,E2 -27387.455} C_VEL
LIN {X 0,Y 139.397,Z 838.41,A -85,B 0,C 180,E1 -27388.836,E2 -27388.836} C_VEL
LIN {X 0,Y 133.758,Z 851.254,A -85,B 0,C 180,E1 -27390.639,E2 -27390.639} C_VEL
LIN {X 0,Y 127.58,Z 862.931,A -85,B 0,C 180,E1 -27392.851,E2 -27392.851} C_VEL
LIN {X 0,Y 121.165,Z 873.657,A -85,B 0,C 180,E1 -27395.703,E2 -27395.703} C_VEL
LIN {X 0,Y 113.75,Z 884.274,A -85,B 0,C 180,E1 -27399.438,E2 -27399.438} C_VEL
LIN {X 0,Y 106.819,Z 893.026,A -85,B 0,C 180,E1 -27403.636,E2 -27403.636} C_VEL
LIN {X 0,Y 99.804,Z 901.438,A -85,B 0,C 180,E1 -27409.355,E2 -27409.355} C_VEL
LIN {X 0,Y 93.869,Z 907.915,A -85,B 0,C 180,E1 -27415.443,E2 -27415.443} C_VEL
LIN {X 0,Y 89.678,Z 912.834,A -85,B 0,C 180,E1 -27421.951,E2 -27421.951} C_VEL
LIN {X 0,Y 85.861,Z 917.638,A -85,B 0,C 180,E1 -27430.888,E2 -27430.888} C_VEL
LIN {X 0,Y 84.093,Z 920.916,A -85,B 0,C 180,E1 -27440.377,E2 -27440.377} C_VEL
LIN {X 0,Y 83.89,Z 922.018,A -85,B 0,C 180,E1 -27445.194,E2 -27445.194} C_VEL
LIN {X 0,Y 84.013,Z 922.771,A -85,B 0,C 180,E1 -27450,E2 -27450} C_VEL
LIN {X 0,Y 84.095,Z 923.21,A -85,B 0,C 180,E1 -27459.621,E2 -27459.621} C_VEL
LIN {X 0,Y 85.939,Z 922.318,A -85,B 0,C 180,E1 -27469.093,E2 -27469.093} C_VEL
LIN {X 0,Y 89.953,Z 920.102,A -85,B 0,C 180,E1 -27477.955,E2 -27477.955} C_VEL
LIN {X 0,Y 95.733,Z 916.503,A -85,B 0,C 180,E1 -27485.965,E2 -27485.965} C_VEL
LIN {X 0,Y 103.188,Z 911.423,A -85,B 0,C 180,E1 -27492.928,E2 -27492.928} C_VEL
LIN {X 0,Y 111.971,Z 904.718,A -85,B 0,C 180,E1 -27498.868,E2 -27498.868} C_VEL
LIN {X 0,Y 120.658,Z 897.276,A -85,B 0,C 180,E1 -27503.216,E2 -27503.216} C_VEL
LIN {X 0,Y 129.504,Z 888.51,A -85,B 0,C 180,E1 -27506.822,E2 -27506.822} C_VEL
LIN {X 0,Y 138.155,Z 878.435,A -85,B 0,C 180,E1 -27509.859,E2 -27509.859} C_VEL
LIN {X 0,Y 146.082,Z 867.792,A -85,B 0,C 180,E1 -27512.131,E2 -27512.131} C_VEL
LIN {X 0,Y 153.374,Z 856.309,A -85,B 0,C 180,E1 -27513.904,E2 -27513.904} C_VEL
LIN {X 0,Y 155.824,Z 851.452,A -85,B 0,C 180,E1 -27514.748,E2 -27514.748} C_VEL
LIN {X 0,Y 158.741,Z 843.404,A -85,B 0,C 180,E1 -27516.578,E2 -27516.578} C_VEL
LIN {X 0,Y 161.478,Z 835.042,A -85,B 0,C 180,E1 -27518.218,E2 -27518.218} C_VEL
LIN {X 0,Y 163.356,Z 829.715,A -85,B 0,C 180,E1 -27518.819,E2 -27518.819} C_VEL
LIN {X 0,Y 167.811,Z 816.147,A -85,B 0,C 180,E1 -27519.579,E2 -27519.579} C_VEL
LIN {X 0,Y 171.168,Z 801.561,A -85,B 0,C 180,E1 -27520.15,E2 -27520.15} C_VEL
LIN {X 0,Y 173.44,Z 784.641,A -85,B 0,C 180,E1 -27520.601,E2 -27520.601} C_VEL
LIN {X 0,Y 173.845,Z 780.391,A -85,B 0,C 180,E1 -27520.751,E2 -27520.751} C_VEL
LIN {X 0,Y 172.205,Z 774.296,A -85,B 0,C 180,E1 -27523.607,E2 -27523.607} C_VEL
LIN {X 0,Y 171.342,Z 771.589,A -85,B 0,C 180,E1 -27525.298,E2 -27525.298} C_VEL
LIN {X 0,Y 169.87,Z 768.303,A -85,B 0,C 180,E1 -27528.591,E2 -27528.591} C_VEL
LIN {X 0,Y 168.822,Z 765.486,A -85,B 0,C 180,E1 -27532.225,E2 -27532.225} C_VEL
LIN {X 0,Y 168.168,Z 764.276,A -85,B 0,C 180,E1 -27537.606,E2 -27537.606} C_VEL
LIN {X 0,Y 168.325,Z 764.664,A -85,B 0,C 180,E1 -27540.599,E2 -27540.599} C_VEL
LIN {X 0,Y 168.983,Z 765.85,A -85,B 0,C 180,E1 -27544.025,E2 -27544.025} C_VEL
LIN {X 0,Y 170.408,Z 769.521,A -85,B 0,C 180,E1 -27548.319,E2 -27548.319} C_VEL
LIN {X 0,Y 172.009,Z 773.324,A -85,B 0,C 180,E1 -27551.542,E2 -27551.542} C_VEL
LIN {X 0,Y 174.055,Z 778.329,A -85,B 0,C 180,E1 -27554.768,E2 -27554.768} C_VEL
LIN {X 0,Y 171.887,Z 795.889,A -85,B 0,C 180,E1 -27555.287,E2 -27555.287} C_VEL
LIN {X 0,Y 168.705,Z 810.519,A -85,B 0,C 180,E1 -27555.89,E2 -27555.89} C_VEL
LIN {X 0,Y 164.276,Z 824.84,A -85,B 0,C 180,E1 -27556.816,E2 -27556.816} C_VEL
LIN {X 0,Y 159.293,Z 836.799,A -85,B 0,C 180,E1 -27557.742,E2 -27557.742} C_VEL
LIN {X 0,Y 153.362,Z 848.558,A -85,B 0,C 180,E1 -27559.063,E2 -27559.063} C_VEL
LIN {X 0,Y 146.53,Z 859.793,A -85,B 0,C 180,E1 -27560.727,E2 -27560.727} C_VEL
LIN {X 0,Y 139.069,Z 870.117,A -85,B 0,C 180,E1 -27562.738,E2 -27562.738} C_VEL
LIN {X 0,Y 130.762,Z 879.936,A -85,B 0,C 180,E1 -27565.328,E2 -27565.328} C_VEL
LIN {X 0,Y 122.066,Z 888.788,A -85,B 0,C 180,E1 -27568.596,E2 -27568.596} C_VEL
LIN {X 0,Y 112.768,Z 896.823,A -85,B 0,C 180,E1 -27572.717,E2 -27572.717} C_VEL
LIN {X 0,Y 105.005,Z 902.704,A -85,B 0,C 180,E1 -27577.041,E2 -27577.041} C_VEL
LIN {X 0,Y 96.381,Z 908.343,A -85,B 0,C 180,E1 -27583.182,E2 -27583.182} C_VEL
LIN {X 0,Y 88.841,Z 912.625,A -85,B 0,C 180,E1 -27590.739,E2 -27590.739} C_VEL
LIN {X 0,Y 82.911,Z 915.448,A -85,B 0,C 180,E1 -27599.43,E2 -27599.43} C_VEL
LIN {X 0,Y 78.84,Z 916.902,A -85,B 0,C 180,E1 -27609.111,E2 -27609.111} C_VEL
LIN {X 0,Y 77.016,Z 917.023,A -85,B 0,C 180,E1 -27619.485,E2 -27619.485} C_VEL
LIN {X 0,Y 76.999,Z 915.841,A -85,B 0,C 180,E1 -27630.001,E2 -27630.001} C_VEL
LIN {X 0,Y 77.629,Z 914.762,A -85,B 0,C 180,E1 -27635.195,E2 -27635.195} C_VEL
LIN {X 0,Y 80.134,Z 911.591,A -85,B 0,C 180,E1 -27645.255,E2 -27645.255} C_VEL
LIN {X 0,Y 84.787,Z 906.931,A -85,B 0,C 180,E1 -27654.485,E2 -27654.485} C_VEL
LIN {X 0,Y 90.941,Z 900.673,A -85,B 0,C 180,E1 -27662.75,E2 -27662.75} C_VEL
LIN {X 0,Y 97.567,Z 893.705,A -85,B 0,C 180,E1 -27669.072,E2 -27669.072} C_VEL
LIN {X 0,Y 104.215,Z 886.401,A -85,B 0,C 180,E1 -27673.728,E2 -27673.728} C_VEL
LIN {X 0,Y 111.407,Z 877.624,A -85,B 0,C 180,E1 -27677.837,E2 -27677.837} C_VEL
LIN {X 0,Y 118.876,Z 867.02,A -85,B 0,C 180,E1 -27681.569,E2 -27681.569} C_VEL
LIN {X 0,Y 124.082,Z 858.622,A -85,B 0,C 180,E1 -27683.816,E2 -27683.816} C_VEL
LIN {X 0,Y 130.211,Z 847.371,A -85,B 0,C 180,E1 -27686.084,E2 -27686.084} C_VEL
LIN {X 0,Y 135.835,Z 835.069,A -85,B 0,C 180,E1 -27687.913,E2 -27687.913} C_VEL
LIN {X 0,Y 140.809,Z 821.361,A -85,B 0,C 180,E1 -27689.427,E2 -27689.427} C_VEL
LIN {X 0,Y 144.535,Z 807.619,A -85,B 0,C 180,E1 -27690.54,E2 -27690.54} C_VEL
LIN {X 0,Y 147.13,Z 793.809,A -85,B 0,C 180,E1 -27691.298,E2 -27691.298} C_VEL
LIN {X 0,Y 150.6,Z 761.102,A -85,B 0,C 180,E1 -27692.331,E2 -27692.331} C_VEL
LIN {X 0,Y 150.715,Z 759.155,A -85,B 0,C 180,E1 -27692.454,E2 -27692.454} C_VEL
LIN {X 0,Y 147.342,Z 751.146,A -85,B 0,C 180,E1 -27696.542,E2 -27696.542} C_VEL
LIN {X 0,Y 144.871,Z 745.981,A -85,B 0,C 180,E1 -27700.148,E2 -27700.148} C_VEL
LIN {X 0,Y 143.211,Z 742.789,A -85,B 0,C 180,E1 -27703.095,E2 -27703.095} C_VEL
LIN {X 0,Y 141.619,Z 739.605,A -85,B 0,C 180,E1 -27706.776,E2 -27706.776} C_VEL
LIN {X 0,Y 140.175,Z 736.252,A -85,B 0,C 180,E1 -27712.435,E2 -27712.435} C_VEL
LIN {X 0,Y 140.054,Z 735.76,A -85,B 0,C 180,E1 -27713.426,E2 -27713.426} C_VEL
LIN {X 0,Y 140.003,Z 735.491,A -85,B 0,C 180,E1 -27720.54,E2 -27720.54} C_VEL
LIN {X 0,Y 140.236,Z 735.927,A -85,B 0,C 180,E1 -27722.181,E2 -27722.181} C_VEL
LIN {X 0,Y 142.112,Z 740.45,A -85,B 0,C 180,E1 -27728.962,E2 -27728.962} C_VEL
LIN {X 0,Y 143.954,Z 744.165,A -85,B 0,C 180,E1 -27732.79,E2 -27732.79} C_VEL
LIN {X 0,Y 146.396,Z 749.072,A -85,B 0,C 180,E1 -27736.65,E2 -27736.65} C_VEL
LIN {X 0,Y 148.491,Z 753.968,A -85,B 0,C 180,E1 -27739.458,E2 -27739.458} C_VEL
LIN {X 0,Y 150.587,Z 761.603,A -85,B 0,C 180,E1 -27742.207,E2 -27742.207} C_VEL
LIN {X 0,Y 147.216,Z 795.546,A -85,B 0,C 180,E1 -27743.32,E2 -27743.32} C_VEL
LIN {X 0,Y 144.67,Z 809.946,A -85,B 0,C 180,E1 -27743.948,E2 -27743.948} C_VEL
LIN {X 0,Y 140.898,Z 824.03,A -85,B 0,C 180,E1 -27744.878,E2 -27744.878} C_VEL
LIN {X 0,Y 136.103,Z 837.54,A -85,B 0,C 180,E1 -27746.207,E2 -27746.207} C_VEL
LIN {X 0,Y 130.265,Z 850.497,A -85,B 0,C 180,E1 -27747.936,E2 -27747.936} C_VEL
LIN {X 0,Y 123.865,Z 862.262,A -85,B 0,C 180,E1 -27750.085,E2 -27750.085} C_VEL
LIN {X 0,Y 117.137,Z 873.052,A -85,B 0,C 180,E1 -27752.862,E2 -27752.862} C_VEL
LIN {X 0,Y 110.585,Z 882.076,A -85,B 0,C 180,E1 -27755.874,E2 -27755.874} C_VEL
LIN {X 0,Y 103.214,Z 891.156,A -85,B 0,C 180,E1 -27760,E2 -27760} C_VEL
LIN {X 0,Y 95.477,Z 899.849,A -85,B 0,C 180,E1 -27765.629,E2 -27765.629} C_VEL
LIN {X 0,Y 89.65,Z 905.943,A -85,B 0,C 180,E1 -27771.159,E2 -27771.159} C_VEL
LIN {X 0,Y 84.782,Z 910.989,A -85,B 0,C 180,E1 -27777.396,E2 -27777.396} C_VEL
LIN {X 0,Y 80.031,Z 916.193,A -85,B 0,C 180,E1 -27786.723,E2 -27786.723} C_VEL
LIN {X 0,Y 77.838,Z 919.118,A -85,B 0,C 180,E1 -27794.283,E2 -27794.283} C_VEL
LIN {X 0,Y 76.795,Z 921.71,A -85,B 0,C 180,E1 -27804.749,E2 -27804.749} C_VEL
LIN {X 0,Y 76.91,Z 922.478,A -85,B 0,C 180,E1 -27809.999,E2 -27809.999} C_VEL
LIN {X 0,Y 77.074,Z 922.943,A -85,B 0,C 180,E1 -27820.507,E2 -27820.507} C_VEL
LIN {X 0,Y 79.209,Z 922.076,A -85,B 0,C 180,E1 -27830.787,E2 -27830.787} C_VEL
LIN {X 0,Y 83.693,Z 919.888,A -85,B 0,C 180,E1 -27840.254,E2 -27840.254} C_VEL
LIN {X 0,Y 90.223,Z 916.208,A -85,B 0,C 180,E1 -27848.836,E2 -27848.836} C_VEL
LIN {X 0,Y 98.068,Z 911.268,A -85,B 0,C 180,E1 -27855.778,E2 -27855.778} C_VEL
LIN {X 0,Y 107.408,Z 904.595,A -85,B 0,C 180,E1 -27861.738,E2 -27861.738} C_VEL
LIN {X 0,Y 116.537,Z 897.2,A -85,B 0,C 180,E1 -27866.018,E2 -27866.018} C_VEL
LIN {X 0,Y 125.486,Z 888.766,A -85,B 0,C 180,E1 -27869.442,E2 -27869.442} C_VEL
LIN {X 0,Y 134.731,Z 878.46,A -85,B 0,C 180,E1 -27872.47,E2 -27872.47} C_VEL
LIN {X 0,Y 142.907,Z 867.878,A -85,B 0,C 180,E1 -27874.643,E2 -27874.643} C_VEL
LIN {X 0,Y 150.557,Z 856.198,A -85,B 0,C 180,E1 -27876.362,E2 -27876.362} C_VEL
LIN {X 0,Y 156.769,Z 844.804,A -85,B 0,C 180,E1 -27877.612,E2 -27877.612} C_VEL
LIN {X 0,Y 162.249,Z 832.477,A -85,B 0,C 180,E1 -27878.638,E2 -27878.638} C_VEL
LIN {X 0,Y 163.356,Z 829.715,A -85,B 0,C 180,E1 -27878.819,E2 -27878.819} C_VEL
LIN {X 0,Y 165.165,Z 824.306,A -85,B 0,C 180,E1 -27879.366,E2 -27879.366} C_VEL
LIN {X 0,Y 167.01,Z 815.445,A -85,B 0,C 180,E1 -27880.785,E2 -27880.785} C_VEL
LIN {X 0,Y 168.352,Z 806.38,A -85,B 0,C 180,E1 -27882.086,E2 -27882.086} C_VEL
LIN {X 0,Y 169.299,Z 800.654,A -85,B 0,C 180,E1 -27882.451,E2 -27882.451} C_VEL
LIN {X 0,Y 171.518,Z 784.098,A -85,B 0,C 180,E1 -27882.892,E2 -27882.892} C_VEL
LIN {X 0,Y 170.375,Z 779.32,A -85,B 0,C 180,E1 -27885.289,E2 -27885.289} C_VEL
LIN {X 0,Y 169.473,Z 776.932,A -85,B 0,C 180,E1 -27887.274,E2 -27887.274} C_VEL
LIN {X 0,Y 168.64,Z 774.874,A -85,B 0,C 180,E1 -27889.495,E2 -27889.495} C_VEL
LIN {X 0,Y 167.816,Z 772.403,A -85,B 0,C 180,E1 -27892.783,E2 -27892.783} C_VEL
LIN {X 0,Y 167.301,Z 771.338,A -85,B 0,C 180,E1 -27897.593,E2 -27897.593} C_VEL
LIN {X 0,Y 167.488,Z 771.846,A -85,B 0,C 180,E1 -27900.902,E2 -27900.902} C_VEL
LIN {X 0,Y 167.988,Z 772.823,A -85,B 0,C 180,E1 -27903.599,E2 -27903.599} C_VEL
LIN {X 0,Y 169.253,Z 776.354,A -85,B 0,C 180,E1 -27907.757,E2 -27907.757} C_VEL
LIN {X 0,Y 170.583,Z 779.796,A -85,B 0,C 180,E1 -27910.685,E2 -27910.685} C_VEL
LIN {X 0,Y 171.659,Z 782.58,A -85,B 0,C 180,E1 -27912.619,E2 -27912.619} C_VEL
LIN {X 0,Y 169.536,Z 798.011,A -85,B 0,C 180,E1 -27913.077,E2 -27913.077} C_VEL
LIN {X 0,Y 166.323,Z 811.846,A -85,B 0,C 180,E1 -27913.623,E2 -27913.623} C_VEL
LIN {X 0,Y 161.947,Z 825.423,A -85,B 0,C 180,E1 -27914.467,E2 -27914.467} C_VEL
LIN {X 0,Y 156.698,Z 837.677,A -85,B 0,C 180,E1 -27915.364,E2 -27915.364} C_VEL
LIN {X 0,Y 150.164,Z 850.097,A -85,B 0,C 180,E1 -27916.713,E2 -27916.713} C_VEL
LIN {X 0,Y 142.604,Z 861.865,A -85,B 0,C 180,E1 -27918.432,E2 -27918.432} C_VEL
LIN {X 0,Y 134.938,Z 871.888,A -85,B 0,C 180,E1 -27920.365,E2 -27920.365} C_VEL
LIN {X 0,Y 126.16,Z 881.659,A -85,B 0,C 180,E1 -27922.952,E2 -27922.952} C_VEL
LIN {X 0,Y 117.364,Z 890.07,A -85,B 0,C 180,E1 -27926.074,E2 -27926.074} C_VEL
LIN {X 0,Y 107.709,Z 897.92,A -85,B 0,C 180,E1 -27930.168,E2 -27930.168} C_VEL
LIN {X 0,Y 98.207,Z 904.517,A -85,B 0,C 180,E1 -27935.32,E2 -27935.32} C_VEL
LIN {X 0,Y 89.415,Z 909.738,A -85,B 0,C 180,E1 -27941.696,E2 -27941.696} C_VEL
LIN {X 0,Y 83.388,Z 912.821,A -85,B 0,C 180,E1 -27947.605,E2 -27947.605} C_VEL
LIN {X 0,Y 76.821,Z 915.673,A -85,B 0,C 180,E1 -27956.708,E2 -27956.708} C_VEL
LIN {X 0,Y 72.181,Z 917.156,A -85,B 0,C 180,E1 -27967.079,E2 -27967.079} C_VEL
LIN {X 0,Y 70,Z 917.305,A -85,B 0,C 180,E1 -27978.417,E2 -27978.417} C_VEL
LIN {X 0,Y 69.725,Z 916.889,A -85,B 0,C 180,E1 -27984.216,E2 -27984.216} C_VEL
LIN {X 0,Y 70.574,Z 915.086,A -85,B 0,C 180,E1 -27995.716,E2 -27995.716} C_VEL
LIN {X 0,Y 73.341,Z 911.95,A -85,B 0,C 180,E1 -28006.708,E2 -28006.708} C_VEL
LIN {X 0,Y 78.397,Z 907.331,A -85,B 0,C 180,E1 -28016.631,E2 -28016.631} C_VEL
LIN {X 0,Y 85.074,Z 901.108,A -85,B 0,C 180,E1 -28025.33,E2 -28025.33} C_VEL
LIN {X 0,Y 92.179,Z 894.179,A -85,B 0,C 180,E1 -28031.846,E2 -28031.846} C_VEL
LIN {X 0,Y 100.495,Z 885.568,A -85,B 0,C 180,E1 -28037.249,E2 -28037.249} C_VEL
LIN {X 0,Y 108.096,Z 876.574,A -85,B 0,C 180,E1 -28041.279,E2 -28041.279} C_VEL
LIN {X 0,Y 115.994,Z 865.706,A -85,B 0,C 180,E1 -28044.882,E2 -28044.882} C_VEL
LIN {X 0,Y 122.841,Z 854.646,A -85,B 0,C 180,E1 -28047.553,E2 -28047.553} C_VEL
LIN {X 0,Y 129.308,Z 842.402,A -85,B 0,C 180,E1 -28049.635,E2 -28049.635} C_VEL
LIN {X 0,Y 135.167,Z 828.671,A -85,B 0,C 180,E1 -28051.333,E2 -28051.333} C_VEL
LIN {X 0,Y 139.56,Z 815.27,A -85,B 0,C 180,E1 -28052.57,E2 -28052.57} C_VEL
LIN {X 0,Y 142.961,Z 801.004,A -85,B 0,C 180,E1 -28053.494,E2 -28053.494} C_VEL
LIN {X 0,Y 145.107,Z 786.75,A -85,B 0,C 180,E1 -28054.098,E2 -28054.098} C_VEL
LIN {X 0,Y 147.545,Z 762.681,A -85,B 0,C 180,E1 -28054.836,E2 -28054.836} C_VEL
LIN {X 0,Y 144.526,Z 755.113,A -85,B 0,C 180,E1 -28059.107,E2 -28059.107} C_VEL
LIN {X 0,Y 142.123,Z 749.86,A -85,B 0,C 180,E1 -28063.405,E2 -28063.405} C_VEL
LIN {X 0,Y 140.505,Z 746.471,A -85,B 0,C 180,E1 -28067.358,E2 -28067.358} C_VEL
LIN {X 0,Y 139.228,Z 743.277,A -85,B 0,C 180,E1 -28072.845,E2 -28072.845} C_VEL
LIN {X 0,Y 139.08,Z 742.754,A -85,B 0,C 180,E1 -28074.199,E2 -28074.199} C_VEL
LIN {X 0,Y 139.214,Z 742.63,A -85,B 0,C 180,E1 -28081.13,E2 -28081.13} C_VEL
LIN {X 0,Y 140.841,Z 747.09,A -85,B 0,C 180,E1 -28088.067,E2 -28088.067} C_VEL
LIN {X 0,Y 142.568,Z 750.884,A -85,B 0,C 180,E1 -28092.002,E2 -28092.002} C_VEL
LIN {X 0,Y 144.596,Z 755.307,A -85,B 0,C 180,E1 -28095.504,E2 -28095.504} C_VEL
LIN {X 0,Y 146.285,Z 759.649,A -85,B 0,C 180,E1 -28098.015,E2 -28098.015} C_VEL
LIN {X 0,Y 147.485,Z 764.643,A -85,B 0,C 180,E1 -28099.847,E2 -28099.847} C_VEL
LIN {X 0,Y 144.044,Z 796.977,A -85,B 0,C 180,E1 -28100.824,E2 -28100.824} C_VEL
LIN {X 0,Y 141.265,Z 811.387,A -85,B 0,C 180,E1 -28101.481,E2 -28101.481} C_VEL
LIN {X 0,Y 137.273,Z 825.288,A -85,B 0,C 180,E1 -28102.378,E2 -28102.378} C_VEL
LIN {X 0,Y 132.349,Z 838.446,A -85,B 0,C 180,E1 -28103.649,E2 -28103.649} C_VEL
LIN {X 0,Y 126.325,Z 851.175,A -85,B 0,C 180,E1 -28105.303,E2 -28105.303} C_VEL
LIN {X 0,Y 119.716,Z 862.773,A -85,B 0,C 180,E1 -28107.385,E2 -28107.385} C_VEL
LIN {X 0,Y 113.389,Z 872.442,A -85,B 0,C 180,E1 -28109.802,E2 -28109.802} C_VEL
LIN {X 0,Y 105.238,Z 883.172,A -85,B 0,C 180,E1 -28113.407,E2 -28113.407} C_VEL
LIN {X 0,Y 97.499,Z 892.017,A -85,B 0,C 180,E1 -28117.541,E2 -28117.541} C_VEL
LIN {X 0,Y 89.388,Z 900.514,A -85,B 0,C 180,E1 -28123.342,E2 -28123.342} C_VEL
LIN {X 0,Y 82.276,Z 907.297,A -85,B 0,C 180,E1 -28130.081,E2 -28130.081} C_VEL
LIN {X 0,Y 77.299,Z 912.04,A -85,B 0,C 180,E1 -28136.939,E2 -28136.939} C_VEL
LIN {X 0,Y 72.483,Z 916.909,A -85,B 0,C 180,E1 -28147.179,E2 -28147.179} C_VEL
LIN {X 0,Y 70.057,Z 920.265,A -85,B 0,C 180,E1 -28158.425,E2 -28158.425} C_VEL
LIN {X 0,Y 69.707,Z 921.401,A -85,B 0,C 180,E1 -28164.213,E2 -28164.213} C_VEL
LIN {X 0,Y 69.815,Z 922.185,A -85,B 0,C 180,E1 -28169.999,E2 -28169.999} C_VEL
LIN {X 0,Y 70.064,Z 922.674,A -85,B 0,C 180,E1 -28181.572,E2 -28181.572} C_VEL
LIN {X 0,Y 72.565,Z 921.835,A -85,B 0,C 180,E1 -28192.793,E2 -28192.793} C_VEL
LIN {X 0,Y 77.59,Z 919.674,A -85,B 0,C 180,E1 -28202.92,E2 -28202.92} C_VEL
LIN {X 0,Y 84.567,Z 916.132,A -85,B 0,C 180,E1 -28211.67,E2 -28211.67} C_VEL
LIN {X 0,Y 93.226,Z 911.113,A -85,B 0,C 180,E1 -28218.926,E2 -28218.926} C_VEL
LIN {X 0,Y 103.136,Z 904.473,A -85,B 0,C 180,E1 -28224.857,E2 -28224.857} C_VEL
LIN {X 0,Y 112.714,Z 897.117,A -85,B 0,C 180,E1 -28229.02,E2 -28229.02} C_VEL
LIN {X 0,Y 121.464,Z 889.256,A -85,B 0,C 180,E1 -28232.146,E2 -28232.146} C_VEL
LIN {X 0,Y 130.088,Z 880.212,A -85,B 0,C 180,E1 -28234.811,E2 -28234.811} C_VEL
LIN {X 0,Y 138.471,Z 870.061,A -85,B 0,C 180,E1 -28236.914,E2 -28236.914} C_VEL
LIN {X 0,Y 146.283,Z 858.923,A -85,B 0,C 180,E1 -28238.568,E2 -28238.568} C_VEL
LIN {X 0,Y 153.418,Z 846.643,A -85,B 0,C 180,E1 -28239.899,E2 -28239.899} C_VEL
LIN {X 0,Y 159.81,Z 832.876,A -85,B 0,C 180,E1 -28240.998,E2 -28240.998} C_VEL
LIN {X 0,Y 164.578,Z 819.681,A -85,B 0,C 180,E1 -28241.743,E2 -28241.743} C_VEL
LIN {X 0,Y 168.31,Z 805.562,A -85,B 0,C 180,E1 -28242.31,E2 -28242.31} C_VEL
LIN {X 0,Y 169.299,Z 800.654,A -85,B 0,C 180,E1 -28242.451,E2 -28242.451} C_VEL
LIN {X 0,Y 169.847,Z 796.655,A -85,B 0,C 180,E1 -28242.759,E2 -28242.759} C_VEL
LIN {X 0,Y 169.92,Z 792.966,A -85,B 0,C 180,E1 -28243.418,E2 -28243.418} C_VEL
LIN {X 0,Y 169.601,Z 788.747,A -85,B 0,C 180,E1 -28244.679,E2 -28244.679} C_VEL
LIN {X 0,Y 168.981,Z 785.555,A -85,B 0,C 180,E1 -28246.261,E2 -28246.261} C_VEL
LIN {X 0,Y 168.6,Z 784.482,A -85,B 0,C 180,E1 -28247.147,E2 -28247.147} C_VEL
LIN {X 0,Y 167.662,Z 781.928,A -85,B 0,C 180,E1 -28249.739,E2 -28249.739} C_VEL
LIN {X 0,Y 166.95,Z 779.497,A -85,B 0,C 180,E1 -28252.745,E2 -28252.745} C_VEL
LIN {X 0,Y 166.433,Z 778.397,A -85,B 0,C 180,E1 -28257.581,E2 -28257.581} C_VEL
LIN {X 0,Y 166.658,Z 779.006,A -85,B 0,C 180,E1 -28261.209,E2 -28261.209} C_VEL
LIN {X 0,Y 167.008,Z 779.758,A -85,B 0,C 180,E1 -28263.167,E2 -28263.167} C_VEL
LIN {X 0,Y 168.12,Z 783.211,A -85,B 0,C 180,E1 -28267.205,E2 -28267.205} C_VEL
LIN {X 0,Y 169.256,Z 786.423,A -85,B 0,C 180,E1 -28269.939,E2 -28269.939} C_VEL
LIN {X 0,Y 169.465,Z 786.986,A -85,B 0,C 180,E1 -28270.379,E2 -28270.379} C_VEL
LIN {X 0,Y 167.199,Z 801.169,A -85,B 0,C 180,E1 -28270.84,E2 -28270.84} C_VEL
LIN {X 0,Y 163.613,Z 815.123,A -85,B 0,C 180,E1 -28271.425,E2 -28271.425} C_VEL
LIN {X 0,Y 159.013,Z 828.132,A -85,B 0,C 180,E1 -28272.173,E2 -28272.173} C_VEL
LIN {X 0,Y 153.339,Z 840.583,A -85,B 0,C 180,E1 -28273.107,E2 -28273.107} C_VEL
LIN {X 0,Y 146.664,Z 852.511,A -85,B 0,C 180,E1 -28274.392,E2 -28274.392} C_VEL
LIN {X 0,Y 138.919,Z 863.906,A -85,B 0,C 180,E1 -28276.009,E2 -28276.009} C_VEL
LIN {X 0,Y 131.054,Z 873.631,A -85,B 0,C 180,E1 -28277.849,E2 -28277.849} C_VEL
LIN {X 0,Y 121.693,Z 883.476,A -85,B 0,C 180,E1 -28280.434,E2 -28280.434} C_VEL
LIN {X 0,Y 112.916,Z 891.355,A -85,B 0,C 180,E1 -28283.357,E2 -28283.357} C_VEL
LIN {X 0,Y 102.871,Z 899.018,A -85,B 0,C 180,E1 -28287.36,E2 -28287.36} C_VEL
LIN {X 0,Y 94.683,Z 904.375,A -85,B 0,C 180,E1 -28291.508,E2 -28291.508} C_VEL
LIN {X 0,Y 84.791,Z 909.901,A -85,B 0,C 180,E1 -28298.055,E2 -28298.055} C_VEL
LIN {X 0,Y 78.217,Z 913.016,A -85,B 0,C 180,E1 -28304.044,E2 -28304.044} C_VEL
LIN {X 0,Y 70.937,Z 915.897,A -85,B 0,C 180,E1 -28313.528,E2 -28313.528} C_VEL
LIN {X 0,Y 65.632,Z 917.41,A -85,B 0,C 180,E1 -28324.639,E2 -28324.639} C_VEL
LIN {X 0,Y 63.024,Z 917.587,A -85,B 0,C 180,E1 -28337.114,E2 -28337.114} C_VEL
LIN {X 0,Y 62.79,Z 916.46,A -85,B 0,C 180,E1 -28350.001,E2 -28350.001} C_VEL
LIN {X 0,Y 63.528,Z 915.409,A -85,B 0,C 180,E1 -28356.352,E2 -28356.352} C_VEL
LIN {X 0,Y 66.597,Z 912.305,A -85,B 0,C 180,E1 -28368.458,E2 -28368.458} C_VEL
LIN {X 0,Y 72.137,Z 907.732,A -85,B 0,C 180,E1 -28379.153,E2 -28379.153} C_VEL
LIN {X 0,Y 79.402,Z 901.544,A -85,B 0,C 180,E1 -28388.286,E2 -28388.286} C_VEL
LIN {X 0,Y 87.038,Z 894.651,A -85,B 0,C 180,E1 -28394.954,E2 -28394.954} C_VEL
LIN {X 0,Y 95.831,Z 886.084,A -85,B 0,C 180,E1 -28400.358,E2 -28400.358} C_VEL
LIN {X 0,Y 103.823,Z 877.138,A -85,B 0,C 180,E1 -28404.323,E2 -28404.323} C_VEL
LIN {X 0,Y 112.083,Z 866.328,A -85,B 0,C 180,E1 -28407.834,E2 -28407.834} C_VEL
LIN {X 0,Y 119.204,Z 855.352,A -85,B 0,C 180,E1 -28410.416,E2 -28410.416} C_VEL
LIN {X 0,Y 125.896,Z 843.239,A -85,B 0,C 180,E1 -28412.401,E2 -28412.401} C_VEL
LIN {X 0,Y 131.935,Z 829.655,A -85,B 0,C 180,E1 -28414.016,E2 -28414.016} C_VEL
LIN {X 0,Y 136.465,Z 816.474,A -85,B 0,C 180,E1 -28415.19,E2 -28415.19} C_VEL
LIN {X 0,Y 140.071,Z 802.02,A -85,B 0,C 180,E1 -28416.114,E2 -28416.114} C_VEL
LIN {X 0,Y 142.333,Z 787.953,A -85,B 0,C 180,E1 -28416.684,E2 -28416.684} C_VEL
LIN {X 0,Y 144.596,Z 766.26,A -85,B 0,C 180,E1 -28417.356,E2 -28417.356} C_VEL
LIN {X 0,Y 142.59,Z 760.915,A -85,B 0,C 180,E1 -28420.627,E2 -28420.627} C_VEL
LIN {X 0,Y 140.637,Z 756.231,A -85,B 0,C 180,E1 -28424.579,E2 -28424.579} C_VEL
LIN {X 0,Y 139.274,Z 753.132,A -85,B 0,C 180,E1 -28428.354,E2 -28428.354} C_VEL
LIN {X 0,Y 138.218,Z 749.802,A -85,B 0,C 180,E1 -28434.162,E2 -28434.162} C_VEL
LIN {X 0,Y 138.308,Z 749.647,A -85,B 0,C 180,E1 -28440.864,E2 -28440.864} C_VEL
LIN {X 0,Y 139.642,Z 753.841,A -85,B 0,C 180,E1 -28447.273,E2 -28447.273} C_VEL
LIN {X 0,Y 141.051,Z 757.226,A -85,B 0,C 180,E1 -28450.859,E2 -28450.859} C_VEL
LIN {X 0,Y 142.857,Z 761.54,A -85,B 0,C 180,E1 -28454.33,E2 -28454.33} C_VEL
LIN {X 0,Y 144.136,Z 765.171,A -85,B 0,C 180,E1 -28456.463,E2 -28456.463} C_VEL
LIN {X 0,Y 144.618,Z 767.342,A -85,B 0,C 180,E1 -28457.316,E2 -28457.316} C_VEL
LIN {X 0,Y 141.305,Z 797.279,A -85,B 0,C 180,E1 -28458.204,E2 -28458.204} C_VEL
LIN {X 0,Y 138.359,Z 811.839,A -85,B 0,C 180,E1 -28458.837,E2 -28458.837} C_VEL
LIN {X 0,Y 134.329,Z 825.361,A -85,B 0,C 180,E1 -28459.651,E2 -28459.651} C_VEL
LIN {X 0,Y 128.873,Z 839.352,A -85,B 0,C 180,E1 -28460.948,E2 -28460.948} C_VEL
LIN {X 0,Y 122.677,Z 851.855,A -85,B 0,C 180,E1 -28462.514,E2 -28462.514} C_VEL
LIN {X 0,Y 115.847,Z 863.283,A -85,B 0,C 180,E1 -28464.494,E2 -28464.494} C_VEL
LIN {X 0,Y 108.722,Z 873.599,A -85,B 0,C 180,E1 -28467.058,E2 -28467.058} C_VEL
LIN {X 0,Y 100.097,Z 884.262,A -85,B 0,C 180,E1 -28470.672,E2 -28470.672} C_VEL
LIN {X 0,Y 92.005,Z 892.877,A -85,B 0,C 180,E1 -28474.798,E2 -28474.798} C_VEL
LIN {X 0,Y 83.47,Z 901.124,A -85,B 0,C 180,E1 -28480.73,E2 -28480.73} C_VEL
LIN {X 0,Y 75.519,Z 908.003,A -85,B 0,C 180,E1 -28488.114,E2 -28488.114} C_VEL
LIN {X 0,Y 69.858,Z 913.031,A -85,B 0,C 180,E1 -28496.404,E2 -28496.404} C_VEL
LIN {X 0,Y 65.944,Z 916.543,A -85,B 0,C 180,E1 -28504.766,E2 -28504.766} C_VEL
LIN {X 0,Y 63.086,Z 919.935,A -85,B 0,C 180,E1 -28517.125,E2 -28517.125} C_VEL
LIN {X 0,Y 62.614,Z 921.088,A -85,B 0,C 180,E1 -28523.555,E2 -28523.555} C_VEL
LIN {X 0,Y 62.71,Z 921.89,A -85,B 0,C 180,E1 -28529.999,E2 -28529.999} C_VEL
LIN {X 0,Y 63.098,Z 922.407,A -85,B 0,C 180,E1 -28542.871,E2 -28542.871} C_VEL
LIN {X 0,Y 66.03,Z 921.593,A -85,B 0,C 180,E1 -28555.197,E2 -28555.197} C_VEL
LIN {X 0,Y 71.686,Z 919.46,A -85,B 0,C 180,E1 -28566.031,E2 -28566.031} C_VEL
LIN {X 0,Y 79.373,Z 915.947,A -85,B 0,C 180,E1 -28575.1,E2 -28575.1} C_VEL
LIN {X 0,Y 88.704,Z 910.958,A -85,B 0,C 180,E1 -28582.4,E2 -28582.4} C_VEL
LIN {X 0,Y 99.199,Z 904.351,A -85,B 0,C 180,E1 -28588.229,E2 -28588.229} C_VEL
LIN {X 0,Y 109.22,Z 897.031,A -85,B 0,C 180,E1 -28592.223,E2 -28592.223} C_VEL
LIN {X 0,Y 119.394,Z 888.212,A -85,B 0,C 180,E1 -28595.517,E2 -28595.517} C_VEL
LIN {X 0,Y 128.771,Z 878.517,A -85,B 0,C 180,E1 -28598.096,E2 -28598.096} C_VEL
LIN {X 0,Y 137.433,Z 868.057,A -85,B 0,C 180,E1 -28599.993,E2 -28599.993} C_VEL
LIN {X 0,Y 145.451,Z 856.53,A -85,B 0,C 180,E1 -28601.487,E2 -28601.487} C_VEL
LIN {X 0,Y 152.756,Z 843.757,A -85,B 0,C 180,E1 -28602.681,E2 -28602.681} C_VEL
LIN {X 0,Y 158.473,Z 831.303,A -85,B 0,C 180,E1 -28603.542,E2 -28603.542} C_VEL
LIN {X 0,Y 163.157,Z 818.268,A -85,B 0,C 180,E1 -28604.186,E2 -28604.186} C_VEL
LIN {X 0,Y 166.819,Z 804.247,A -85,B 0,C 180,E1 -28604.699,E2 -28604.699} C_VEL
LIN {X 0,Y 169.187,Z 789.95,A -85,B 0,C 180,E1 -28605.051,E2 -28605.051} C_VEL
LIN {X 0,Y 169.383,Z 787.615,A -85,B 0,C 180,E1 -28605.211,E2 -28605.211} C_VEL
LIN {X 0,Y 168.639,Z 784.567,A -85,B 0,C 180,E1 -28607.056,E2 -28607.056} C_VEL
LIN {X 0,Y 168.6,Z 784.482,A -85,B 0,C 180,E1 -28607.147,E2 -28607.147} C_VEL
LIN {X 0,Y 167.755,Z 783.376,A -85,B 0,C 180,E1 -28609.108,E2 -28609.108} C_VEL
LIN {X 0,Y 166.96,Z 783.347,A -85,B 0,C 180,E1 -28611.129,E2 -28611.129} C_VEL
LIN {X 0,Y 165.624,Z 785.254,A -85,B 0,C 180,E1 -28616.641,E2 -28616.641} C_VEL
LIN {X 0,Y 165.564,Z 785.478,A -85,B 0,C 180,E1 -28618.041,E2 -28618.041} C_VEL
LIN {X 0,Y 165.992,Z 786.453,A -85,B 0,C 180,E1 -28622.427,E2 -28622.427} C_VEL
LIN {X 0,Y 166.892,Z 789.904,A -85,B 0,C 180,E1 -28626.499,E2 -28626.499} C_VEL
LIN {X 0,Y 167.428,Z 791.624,A -85,B 0,C 180,E1 -28628.119,E2 -28628.119} C_VEL
LIN {X 0,Y 164.911,Z 804.927,A -85,B 0,C 180,E1 -28628.56,E2 -28628.56} C_VEL
LIN {X 0,Y 160.974,Z 818.797,A -85,B 0,C 180,E1 -28629.162,E2 -28629.162} C_VEL
LIN {X 0,Y 156.041,Z 831.569,A -85,B 0,C 180,E1 -28629.859,E2 -28629.859} C_VEL
LIN {X 0,Y 149.664,Z 844.508,A -85,B 0,C 180,E1 -28630.827,E2 -28630.827} C_VEL
LIN {X 0,Y 142.011,Z 857,A -85,B 0,C 180,E1 -28632.202,E2 -28632.202} C_VEL
LIN {X 0,Y 133.86,Z 867.934,A -85,B 0,C 180,E1 -28633.762,E2 -28633.762} C_VEL
LIN {X 0,Y 124.259,Z 878.703,A -85,B 0,C 180,E1 -28635.95,E2 -28635.95} C_VEL
LIN {X 0,Y 114.881,Z 887.566,A -85,B 0,C 180,E1 -28638.518,E2 -28638.518} C_VEL
LIN {X 0,Y 104.22,Z 896.031,A -85,B 0,C 180,E1 -28641.995,E2 -28641.995} C_VEL
LIN {X 0,Y 94.007,Z 902.82,A -85,B 0,C 180,E1 -28646.217,E2 -28646.217} C_VEL
LIN {X 0,Y 85.746,Z 907.471,A -85,B 0,C 180,E1 -28650.616,E2 -28650.616} C_VEL
LIN {X 0,Y 75.688,Z 912.267,A -85,B 0,C 180,E1 -28657.883,E2 -28657.883} C_VEL
LIN {X 0,Y 67.38,Z 915.481,A -85,B 0,C 180,E1 -28666.9,E2 -28666.9} C_VEL
LIN {X 0,Y 61.976,Z 917.06,A -85,B 0,C 180,E1 -28675.46,E2 -28675.46} C_VEL
LIN {X 0,Y 57.291,Z 917.931,A -85,B 0,C 180,E1 -28688.407,E2 -28688.407} C_VEL
LIN {X 0,Y 55.552,Z 917.481,A -85,B 0,C 180,E1 -28702.733,E2 -28702.733} C_VEL
LIN {X 0,Y 56.478,Z 915.733,A -85,B 0,C 180,E1 -28717.149,E2 -28717.149} C_VEL
LIN {X 0,Y 59.916,Z 912.658,A -85,B 0,C 180,E1 -28730.604,E2 -28730.604} C_VEL
LIN {X 0,Y 66.036,Z 908.131,A -85,B 0,C 180,E1 -28742.151,E2 -28742.151} C_VEL
LIN {X 0,Y 73.984,Z 901.978,A -85,B 0,C 180,E1 -28751.679,E2 -28751.679} C_VEL
LIN {X 0,Y 82.189,Z 895.124,A -85,B 0,C 180,E1 -28758.437,E2 -28758.437} C_VEL
LIN {X 0,Y 91.485,Z 886.599,A -85,B 0,C 180,E1 -28763.769,E2 -28763.769} C_VEL
LIN {X 0,Y 99.871,Z 877.7,A -85,B 0,C 180,E1 -28767.614,E2 -28767.614} C_VEL
LIN {X 0,Y 108.491,Z 866.946,A -85,B 0,C 180,E1 -28770.99,E2 -28770.99} C_VEL
LIN {X 0,Y 115.883,Z 856.039,A -85,B 0,C 180,E1 -28773.452,E2 -28773.452} C_VEL
LIN {X 0,Y 122.793,Z 844.041,A -85,B 0,C 180,E1 -28775.314,E2 -28775.314} C_VEL
LIN {X 0,Y 129.005,Z 830.625,A -85,B 0,C 180,E1 -28776.828,E2 -28776.828} C_VEL
LIN {X 0,Y 133.664,Z 817.657,A -85,B 0,C 180,E1 -28777.93,E2 -28777.93} C_VEL
LIN {X 0,Y 137.416,Z 803.387,A -85,B 0,C 180,E1 -28778.802,E2 -28778.802} C_VEL
LIN {X 0,Y 139.793,Z 789.656,A -85,B 0,C 180,E1 -28779.346,E2 -28779.346} C_VEL
LIN {X 0,Y 141.931,Z 770.053,A -85,B 0,C 180,E1 -28779.945,E2 -28779.945} C_VEL
LIN {X 0,Y 140.295,Z 765.369,A -85,B 0,C 180,E1 -28783.182,E2 -28783.182} C_VEL
LIN {X 0,Y 139.017,Z 762.198,A -85,B 0,C 180,E1 -28786.291,E2 -28786.291} C_VEL
LIN {X 0,Y 138.155,Z 759.924,A -85,B 0,C 180,E1 -28789.118,E2 -28789.118} C_VEL
LIN {X 0,Y 137.279,Z 756.783,A -85,B 0,C 180,E1 -28794.859,E2 -28794.859} C_VEL
LIN {X 0,Y 137.388,Z 756.628,A -85,B 0,C 180,E1 -28800.434,E2 -28800.434} C_VEL
LIN {X 0,Y 138.502,Z 760.687,A -85,B 0,C 180,E1 -28806.578,E2 -28806.578} C_VEL
LIN {X 0,Y 139.79,Z 764.114,A -85,B 0,C 180,E1 -28810.18,E2 -28810.18} C_VEL
LIN {X 0,Y 141.484,Z 768.67,A -85,B 0,C 180,E1 -28813.715,E2 -28813.715} C_VEL
LIN {X 0,Y 142.011,Z 770.289,A -85,B 0,C 180,E1 -28814.691,E2 -28814.691} C_VEL
LIN {X 0,Y 139.229,Z 795.237,A -85,B 0,C 180,E1 -28815.415,E2 -28815.415} C_VEL
LIN {X 0,Y 136.351,Z 810.018,A -85,B 0,C 180,E1 -28815.967,E2 -28815.967} C_VEL
LIN {X 0,Y 132.729,Z 822.54,A -85,B 0,C 180,E1 -28816.625,E2 -28816.625} C_VEL
LIN {X 0,Y 128.092,Z 834.874,A -85,B 0,C 180,E1 -28817.576,E2 -28817.576} C_VEL
LIN {X 0,Y 121.705,Z 848.219,A -85,B 0,C 180,E1 -28818.986,E2 -28818.986} C_VEL
LIN {X 0,Y 114.628,Z 860.241,A -85,B 0,C 180,E1 -28820.771,E2 -28820.771} C_VEL
LIN {X 0,Y 108.494,Z 869.229,A -85,B 0,C 180,E1 -28822.618,E2 -28822.618} C_VEL
LIN {X 0,Y 99.544,Z 880.425,A -85,B 0,C 180,E1 -28825.818,E2 -28825.818} C_VEL
LIN {X 0,Y 90.919,Z 889.643,A -85,B 0,C 180,E1 -28829.584,E2 -28829.584} C_VEL
LIN {X 0,Y 82.787,Z 897.323,A -85,B 0,C 180,E1 -28834.135,E2 -28834.135} C_VEL
LIN {X 0,Y 74.163,Z 904.658,A -85,B 0,C 180,E1 -28840.701,E2 -28840.701} C_VEL
LIN {X 0,Y 67.618,Z 909.793,A -85,B 0,C 180,E1 -28847.499,E2 -28847.499} C_VEL
LIN {X 0,Y 60.896,Z 915.097,A -85,B 0,C 180,E1 -28858.711,E2 -28858.711} C_VEL
LIN {X 0,Y 57.464,Z 918.07,A -85,B 0,C 180,E1 -28868.474,E2 -28868.474} C_VEL
LIN {X 0,Y 55.549,Z 920.773,A -85,B 0,C 180,E1 -28882.731,E2 -28882.731} C_VEL
LIN {X 0,Y 55.604,Z 921.592,A -85,B 0,C 180,E1 -28889.999,E2 -28889.999} C_VEL
LIN {X 0,Y 55.539,Z 922.034,A -85,B 0,C 180,E1 -28897.269,E2 -28897.269} C_VEL
LIN {X 0,Y 57.519,Z 921.91,A -85,B 0,C 180,E1 -28911.503,E2 -28911.503} C_VEL
LIN {X 0,Y 62.535,Z 920.467,A -85,B 0,C 180,E1 -28924.188,E2 -28924.188} C_VEL
LIN {X 0,Y 70.062,Z 917.681,A -85,B 0,C 180,E1 -28934.601,E2 -28934.601} C_VEL
LIN {X 0,Y 79.347,Z 913.475,A -85,B 0,C 180,E1 -28942.859,E2 -28942.859} C_VEL
LIN {X 0,Y 89.988,Z 907.732,A -85,B 0,C 180,E1 -28949.214,E2 -28949.214} C_VEL
LIN {X 0,Y 100.062,Z 901.29,A -85,B 0,C 180,E1 -28953.574,E2 -28953.574} C_VEL
LIN {X 0,Y 110.65,Z 893.312,A -85,B 0,C 180,E1 -28957.069,E2 -28957.069} C_VEL
LIN {X 0,Y 119.972,Z 884.988,A -85,B 0,C 180,E1 -28959.6,E2 -28959.6} C_VEL
LIN {X 0,Y 129.505,Z 874.986,A -85,B 0,C 180,E1 -28961.748,E2 -28961.748} C_VEL
LIN {X 0,Y 138.432,Z 863.87,A -85,B 0,C 180,E1 -28963.387,E2 -28963.387} C_VEL
LIN {X 0,Y 146.65,Z 851.426,A -85,B 0,C 180,E1 -28964.679,E2 -28964.679} C_VEL
LIN {X 0,Y 153.28,Z 839.108,A -85,B 0,C 180,E1 -28965.603,E2 -28965.603} C_VEL
LIN {X 0,Y 159.105,Z 825.393,A -85,B 0,C 180,E1 -28966.357,E2 -28966.357} C_VEL
LIN {X 0,Y 163.548,Z 811.533,A -85,B 0,C 180,E1 -28966.866,E2 -28966.866} C_VEL
LIN {X 0,Y 166.535,Z 798.08,A -85,B 0,C 180,E1 -28967.238,E2 -28967.238} C_VEL
LIN {X 0,Y 167.478,Z 791.698,A -85,B 0,C 180,E1 -28967.447,E2 -28967.447} C_VEL
LIN {X 0,Y 166.553,Z 788.642,A -85,B 0,C 180,E1 -28970.437,E2 -28970.437} C_VEL
LIN {X 0,Y 165.878,Z 786.274,A -85,B 0,C 180,E1 -28973.768,E2 -28973.768} C_VEL
LIN {X 0,Y 165.564,Z 785.478,A -85,B 0,C 180,E1 -28978.041,E2 -28978.041} C_VEL
LIN {X 0,Y 165.521,Z 786.354,A -85,B 0,C 180,E1 -28979.363,E2 -28979.363} C_VEL
LIN {X 0,Y 165.286,Z 789.912,A -85,B 0,C 180,E1 -28981.324,E2 -28981.324} C_VEL
LIN {X 0,Y 165.138,Z 793.894,A -85,B 0,C 180,E1 -28983.266,E2 -28983.266} C_VEL
LIN {X 0,Y 165.254,Z 795.39,A -85,B 0,C 180,E1 -28984.574,E2 -28984.574} C_VEL
LIN {X 0,Y 165.491,Z 796.621,A -85,B 0,C 180,E1 -28985.861,E2 -28985.861} C_VEL
LIN {X 0,Y 162.225,Z 810.81,A -85,B 0,C 180,E1 -28986.304,E2 -28986.304} C_VEL
LIN {X 0,Y 157.597,Z 824.824,A -85,B 0,C 180,E1 -28986.961,E2 -28986.961} C_VEL
LIN {X 0,Y 151.586,Z 838.39,A -85,B 0,C 180,E1 -28987.688,E2 -28987.688} C_VEL
LIN {X 0,Y 144.672,Z 850.75,A -85,B 0,C 180,E1 -28988.708,E2 -28988.708} C_VEL
LIN {X 0,Y 136.498,Z 862.622,A -85,B 0,C 180,E1 -28990.033,E2 -28990.033} C_VEL
LIN {X 0,Y 127.393,Z 873.548,A -85,B 0,C 180,E1 -28991.698,E2 -28991.698} C_VEL
LIN {X 0,Y 117.35,Z 883.586,A -85,B 0,C 180,E1 -28993.862,E2 -28993.862} C_VEL
LIN {X 0,Y 108.029,Z 891.468,A -85,B 0,C 180,E1 -28996.346,E2 -28996.346} C_VEL
LIN {X 0,Y 97.109,Z 899.212,A -85,B 0,C 180,E1 -28999.808,E2 -28999.808} C_VEL
LIN {X 0,Y 87.799,Z 904.76,A -85,B 0,C 180,E1 -29003.594,E2 -29003.594} C_VEL
LIN {X 0,Y 76.772,Z 910.231,A -85,B 0,C 180,E1 -29009.581,E2 -29009.581} C_VEL
LIN {X 0,Y 68.982,Z 913.409,A -85,B 0,C 180,E1 -29015.408,E2 -29015.408} C_VEL
LIN {X 0,Y 60.006,Z 916.348,A -85,B 0,C 180,E1 -29025.354,E2 -29025.354} C_VEL
LIN {X 0,Y 53.04,Z 917.918,A -85,B 0,C 180,E1 -29037.994,E2 -29037.994} C_VEL
LIN {X 0,Y 49.181,Z 918.152,A -85,B 0,C 180,E1 -29053.394,E2 -29053.394} C_VEL
LIN {X 0,Y 48.485,Z 917.777,A -85,B 0,C 180,E1 -29061.666,E2 -29061.666} C_VEL
LIN {X 0,Y 49.453,Z 916.055,A -85,B 0,C 180,E1 -29078.171,E2 -29078.171} C_VEL
LIN {X 0,Y 53.347,Z 913.009,A -85,B 0,C 180,E1 -29093.281,E2 -29093.281} C_VEL
LIN {X 0,Y 60.172,Z 908.522,A -85,B 0,C 180,E1 -29105.733,E2 -29105.733} C_VEL
LIN {X 0,Y 68.859,Z 902.41,A -85,B 0,C 180,E1 -29115.598,E2 -29115.598} C_VEL
LIN {X 0,Y 77.684,Z 895.591,A -85,B 0,C 180,E1 -29122.337,E2 -29122.337} C_VEL
LIN {X 0,Y 87.495,Z 887.108,A -85,B 0,C 180,E1 -29127.503,E2 -29127.503} C_VEL
LIN {X 0,Y 96.278,Z 878.257,A -85,B 0,C 180,E1 -29131.16,E2 -29131.16} C_VEL
LIN {X 0,Y 105.251,Z 867.559,A -85,B 0,C 180,E1 -29134.35,E2 -29134.35} C_VEL
LIN {X 0,Y 112.906,Z 856.722,A -85,B 0,C 180,E1 -29136.657,E2 -29136.657} C_VEL
LIN {X 0,Y 120.017,Z 844.817,A -85,B 0,C 180,E1 -29138.376,E2 -29138.376} C_VEL
LIN {X 0,Y 126.401,Z 831.592,A -85,B 0,C 180,E1 -29139.763,E2 -29139.763} C_VEL
LIN {X 0,Y 131.187,Z 818.838,A -85,B 0,C 180,E1 -29140.773,E2 -29140.773} C_VEL
LIN {X 0,Y 135.087,Z 804.709,A -85,B 0,C 180,E1 -29141.592,E2 -29141.592} C_VEL
LIN {X 0,Y 137.633,Z 790.76,A -85,B 0,C 180,E1 -29142.137,E2 -29142.137} C_VEL
LIN {X 0,Y 139.558,Z 774.018,A -85,B 0,C 180,E1 -29142.603,E2 -29142.603} C_VEL
LIN {X 0,Y 138.085,Z 769.555,A -85,B 0,C 180,E1 -29146.314,E2 -29146.314} C_VEL
LIN {X 0,Y 137.06,Z 766.718,A -85,B 0,C 180,E1 -29149.893,E2 -29149.893} C_VEL
LIN {X 0,Y 136.411,Z 763.867,A -85,B 0,C 180,E1 -29154.826,E2 -29154.826} C_VEL
LIN {X 0,Y 136.474,Z 763.83,A -85,B 0,C 180,E1 -29160.218,E2 -29160.218} C_VEL
LIN {X 0,Y 137.385,Z 767.514,A -85,B 0,C 180,E1 -29165.871,E2 -29165.871} C_VEL
LIN {X 0,Y 138.563,Z 770.98,A -85,B 0,C 180,E1 -29169.51,E2 -29169.51} C_VEL
LIN {X 0,Y 139.602,Z 774.141,A -85,B 0,C 180,E1 -29171.984,E2 -29171.984} C_VEL
LIN {X 0,Y 137.716,Z 791.332,A -85,B 0,C 180,E1 -29172.515,E2 -29172.515} C_VEL
LIN {X 0,Y 135.35,Z 805.113,A -85,B 0,C 180,E1 -29172.938,E2 -29172.938} C_VEL
LIN {X 0,Y 131.88,Z 818.292,A -85,B 0,C 180,E1 -29173.522,E2 -29173.522} C_VEL
LIN {X 0,Y 127.772,Z 829.916,A -85,B 0,C 180,E1 -29174.197,E2 -29174.197} C_VEL
LIN {X 0,Y 122.022,Z 842.719,A -85,B 0,C 180,E1 -29175.259,E2 -29175.259} C_VEL
LIN {X 0,Y 114.704,Z 855.761,A -85,B 0,C 180,E1 -29176.791,E2 -29176.791} C_VEL
LIN {X 0,Y 106.715,Z 867.498,A -85,B 0,C 180,E1 -29178.789,E2 -29178.789} C_VEL
LIN {X 0,Y 98.208,Z 878.138,A -85,B 0,C 180,E1 -29181.515,E2 -29181.515} C_VEL
LIN {X 0,Y 89.093,Z 887.717,A -85,B 0,C 180,E1 -29184.882,E2 -29184.882} C_VEL
LIN {X 0,Y 80.37,Z 895.656,A -85,B 0,C 180,E1 -29189.018,E2 -29189.018} C_VEL
LIN {X 0,Y 72.266,Z 902.271,A -85,B 0,C 180,E1 -29194.243,E2 -29194.243} C_VEL
LIN {X 0,Y 64.357,Z 908.017,A -85,B 0,C 180,E1 -29200.934,E2 -29200.934} C_VEL
LIN {X 0,Y 56.61,Z 913.532,A -85,B 0,C 180,E1 -29211.629,E2 -29211.629} C_VEL
LIN {X 0,Y 50.89,Z 917.72,A -85,B 0,C 180,E1 -29225.524,E2 -29225.524} C_VEL
LIN {X 0,Y 48.489,Z 920.453,A -85,B 0,C 180,E1 -29241.665,E2 -29241.665} C_VEL
LIN {X 0,Y 48.493,Z 921.289,A -85,B 0,C 180,E1 -29249.999,E2 -29249.999} C_VEL
LIN {X 0,Y 48.483,Z 921.747,A -85,B 0,C 180,E1 -29258.334,E2 -29258.334} C_VEL
LIN {X 0,Y 50.944,Z 921.654,A -85,B 0,C 180,E1 -29274.447,E2 -29274.447} C_VEL
LIN {X 0,Y 56.767,Z 920.24,A -85,B 0,C 180,E1 -29288.244,E2 -29288.244} C_VEL
LIN {X 0,Y 65.147,Z 917.483,A -85,B 0,C 180,E1 -29299.038,E2 -29299.038} C_VEL
LIN {X 0,Y 75.252,Z 913.308,A -85,B 0,C 180,E1 -29307.195,E2 -29307.195} C_VEL
LIN {X 0,Y 86.542,Z 907.596,A -85,B 0,C 180,E1 -29313.291,E2 -29313.291} C_VEL
LIN {X 0,Y 97.101,Z 901.19,A -85,B 0,C 180,E1 -29317.341,E2 -29317.341} C_VEL
LIN {X 0,Y 108.081,Z 893.251,A -85,B 0,C 180,E1 -29320.539,E2 -29320.539} C_VEL
LIN {X 0,Y 117.679,Z 884.97,A -85,B 0,C 180,E1 -29322.852,E2 -29322.852} C_VEL
LIN {X 0,Y 127.461,Z 875.019,A -85,B 0,C 180,E1 -29324.779,E2 -29324.779} C_VEL
LIN {X 0,Y 136.577,Z 863.972,A -85,B 0,C 180,E1 -29326.233,E2 -29326.233} C_VEL
LIN {X 0,Y 144.942,Z 851.644,A -85,B 0,C 180,E1 -29327.377,E2 -29327.377} C_VEL
LIN {X 0,Y 151.672,Z 839.444,A -85,B 0,C 180,E1 -29328.198,E2 -29328.198} C_VEL
LIN {X 0,Y 157.588,Z 825.898,A -85,B 0,C 180,E1 -29328.854,E2 -29328.854} C_VEL
LIN {X 0,Y 162.358,Z 811.331,A -85,B 0,C 180,E1 -29329.335,E2 -29329.335} C_VEL
LIN {X 0,Y 165.471,Z 797.486,A -85,B 0,C 180,E1 -29329.666,E2 -29329.666} C_VEL
LIN {X 0,Y 165.601,Z 796.558,A -85,B 0,C 180,E1 -29329.787,E2 -29329.787} C_VEL
LIN {X 0,Y 165.102,Z 794.569,A -85,B 0,C 180,E1 -29332.203,E2 -29332.203} C_VEL
LIN {X 0,Y 164.881,Z 793.294,A -85,B 0,C 180,E1 -29333.884,E2 -29333.884} C_VEL
LIN {X 0,Y 164.6,Z 792.531,A -85,B 0,C 180,E1 -29338.359,E2 -29338.359} C_VEL
LIN {X 0,Y 164.92,Z 793.513,A -85,B 0,C 180,E1 -29342.138,E2 -29342.138} C_VEL
LIN {X 0,Y 165.254,Z 795.39,A -85,B 0,C 180,E1 -29344.574,E2 -29344.574} C_VEL
LIN {X 0,Y 165.211,Z 796.486,A -85,B 0,C 180,E1 -29345.043,E2 -29345.043} C_VEL
LIN {X 0,Y 164.842,Z 798.795,A -85,B 0,C 180,E1 -29345.279,E2 -29345.279} C_VEL
LIN {X 0,Y 163.971,Z 802.513,A -85,B 0,C 180,E1 -29345.124,E2 -29345.124} C_VEL
LIN {X 0,Y 161.335,Z 811.291,A -85,B 0,C 180,E1 -29344.121,E2 -29344.121} C_VEL
LIN {X 0,Y 160.088,Z 815.171,A -85,B 0,C 180,E1 -29343.982,E2 -29343.982} C_VEL
LIN {X 0,Y 159.836,Z 815.926,A -85,B 0,C 180,E1 -29344.006,E2 -29344.006} C_VEL
LIN {X 0,Y 154.672,Z 829.706,A -85,B 0,C 180,E1 -29344.588,E2 -29344.588} C_VEL
LIN {X 0,Y 149.078,Z 841.308,A -85,B 0,C 180,E1 -29345.194,E2 -29345.194} C_VEL
LIN {X 0,Y 142.425,Z 852.597,A -85,B 0,C 180,E1 -29346.065,E2 -29346.065} C_VEL
LIN {X 0,Y 133.739,Z 864.662,A -85,B 0,C 180,E1 -29347.305,E2 -29347.305} C_VEL
LIN {X 0,Y 124.455,Z 875.292,A -85,B 0,C 180,E1 -29348.802,E2 -29348.802} C_VEL
LIN {X 0,Y 114.44,Z 884.854,A -85,B 0,C 180,E1 -29350.708,E2 -29350.708} C_VEL
LIN {X 0,Y 102.973,Z 893.956,A -85,B 0,C 180,E1 -29353.45,E2 -29353.45} C_VEL
LIN {X 0,Y 91.743,Z 901.248,A -85,B 0,C 180,E1 -29356.752,E2 -29356.752} C_VEL
LIN {X 0,Y 82.419,Z 906.332,A -85,B 0,C 180,E1 -29360.285,E2 -29360.285} C_VEL
LIN {X 0,Y 70.601,Z 911.578,A -85,B 0,C 180,E1 -29366.376,E2 -29366.376} C_VEL
LIN {X 0,Y 59.902,Z 915.267,A -85,B 0,C 180,E1 -29374.789,E2 -29374.789} C_VEL
LIN {X 0,Y 50.795,Z 917.542,A -85,B 0,C 180,E1 -29386.228,E2 -29386.228} C_VEL
LIN {X 0,Y 44.263,Z 918.469,A -85,B 0,C 180,E1 -29401.555,E2 -29401.555} C_VEL
LIN {X 0,Y 41.436,Z 918.073,A -85,B 0,C 180,E1 -29420.236,E2 -29420.236} C_VEL
LIN {X 0,Y 42.441,Z 916.378,A -85,B 0,C 180,E1 -29439.533,E2 -29439.533} C_VEL
LIN {X 0,Y 46.927,Z 913.36,A -85,B 0,C 180,E1 -29456.699,E2 -29456.699} C_VEL
LIN {X 0,Y 54.575,Z 908.908,A -85,B 0,C 180,E1 -29470.083,E2 -29470.083} C_VEL
LIN {X 0,Y 61.574,Z 904.5,A -85,B 0,C 180,E1 -29477.895,E2 -29477.895} C_VEL
LIN {X 0,Y 69.398,Z 899.141,A -85,B 0,C 180,E1 -29484.114,E2 -29484.114} C_VEL
LIN {X 0,Y 79.387,Z 891.455,A -85,B 0,C 180,E1 -29489.673,E2 -29489.673} C_VEL
LIN {X 0,Y 88.48,Z 883.417,A -85,B 0,C 180,E1 -29493.329,E2 -29493.329} C_VEL
LIN {X 0,Y 97.723,Z 873.753,A -85,B 0,C 180,E1 -29496.486,E2 -29496.486} C_VEL
LIN {X 0,Y 106.343,Z 863.039,A -85,B 0,C 180,E1 -29498.988,E2 -29498.988} C_VEL
LIN {X 0,Y 113.515,Z 852.443,A -85,B 0,C 180,E1 -29500.766,E2 -29500.766} C_VEL
LIN {X 0,Y 120.857,Z 839.439,A -85,B 0,C 180,E1 -29502.221,E2 -29502.221} C_VEL
LIN {X 0,Y 126.593,Z 826.642,A -85,B 0,C 180,E1 -29503.269,E2 -29503.269} C_VEL
LIN {X 0,Y 131.07,Z 813.57,A -85,B 0,C 180,E1 -29504.116,E2 -29504.116} C_VEL
LIN {X 0,Y 134.553,Z 799.352,A -85,B 0,C 180,E1 -29504.734,E2 -29504.734} C_VEL
LIN {X 0,Y 136.802,Z 784.233,A -85,B 0,C 180,E1 -29505.167,E2 -29505.167} C_VEL
LIN {X 0,Y 137.441,Z 778.238,A -85,B 0,C 180,E1 -29505.394,E2 -29505.394} C_VEL
LIN {X 0,Y 136.364,Z 774.745,A -85,B 0,C 180,E1 -29508.973,E2 -29508.973} C_VEL
LIN {X 0,Y 135.982,Z 773.495,A -85,B 0,C 180,E1 -29510.718,E2 -29510.718} C_VEL
LIN {X 0,Y 135.493,Z 770.84,A -85,B 0,C 180,E1 -29515.537,E2 -29515.537} C_VEL
LIN {X 0,Y 135.561,Z 770.882,A -85,B 0,C 180,E1 -29519.813,E2 -29519.813} C_VEL
LIN {X 0,Y 136.252,Z 774.214,A -85,B 0,C 180,E1 -29524.993,E2 -29524.993} C_VEL
LIN {X 0,Y 137.193,Z 777.402,A -85,B 0,C 180,E1 -29528.376,E2 -29528.376} C_VEL
LIN {X 0,Y 137.503,Z 778.428,A -85,B 0,C 180,E1 -29529.271,E2 -29529.271} C_VEL
LIN {X 0,Y 135.244,Z 796.608,A -85,B 0,C 180,E1 -29529.738,E2 -29529.738} C_VEL
LIN {X 0,Y 132.087,Z 811.158,A -85,B 0,C 180,E1 -29530.198,E2 -29530.198} C_VEL
LIN {X 0,Y 127.878,Z 824.466,A -85,B 0,C 180,E1 -29530.768,E2 -29530.768} C_VEL
LIN {X 0,Y 122.019,Z 838.474,A -85,B 0,C 180,E1 -29531.717,E2 -29531.717} C_VEL
LIN {X 0,Y 115.335,Z 850.986,A -85,B 0,C 180,E1 -29532.846,E2 -29532.846} C_VEL
LIN {X 0,Y 107.071,Z 863.598,A -85,B 0,C 180,E1 -29534.493,E2 -29534.493} C_VEL
LIN {X 0,Y 98.457,Z 874.564,A -85,B 0,C 180,E1 -29536.749,E2 -29536.749} C_VEL
LIN {X 0,Y 89.45,Z 884.181,A -85,B 0,C 180,E1 -29539.466,E2 -29539.466} C_VEL
LIN {X 0,Y 80.16,Z 892.675,A -85,B 0,C 180,E1 -29542.986,E2 -29542.986} C_VEL
LIN {X 0,Y 69.89,Z 900.797,A -85,B 0,C 180,E1 -29548.37,E2 -29548.37} C_VEL
LIN {X 0,Y 60.369,Z 907.336,A -85,B 0,C 180,E1 -29555.419,E2 -29555.419} C_VEL
LIN {X 0,Y 51.174,Z 913.147,A -85,B 0,C 180,E1 -29566.631,E2 -29566.631} C_VEL
LIN {X 0,Y 44.479,Z 917.367,A -85,B 0,C 180,E1 -29581.703,E2 -29581.703} C_VEL
LIN {X 0,Y 41.446,Z 920.13,A -85,B 0,C 180,E1 -29600.236,E2 -29600.236} C_VEL
LIN {X 0,Y 41.402,Z 920.984,A -85,B 0,C 180,E1 -29609.999,E2 -29609.999} C_VEL
LIN {X 0,Y 42.495,Z 921.592,A -85,B 0,C 180,E1 -29629.315,E2 -29629.315} C_VEL
LIN {X 0,Y 47.505,Z 920.867,A -85,B 0,C 180,E1 -29646.282,E2 -29646.282} C_VEL
LIN {X 0,Y 55.775,Z 918.82,A -85,B 0,C 180,E1 -29659.115,E2 -29659.115} C_VEL
LIN {X 0,Y 66.013,Z 915.396,A -85,B 0,C 180,E1 -29668.397,E2 -29668.397} C_VEL
LIN {X 0,Y 77.509,Z 910.502,A -85,B 0,C 180,E1 -29675.057,E2 -29675.057} C_VEL
LIN {X 0,Y 89.811,Z 903.996,A -85,B 0,C 180,E1 -29679.89,E2 -29679.89} C_VEL
LIN {X 0,Y 101.029,Z 896.786,A -85,B 0,C 180,E1 -29683.038,E2 -29683.038} C_VEL
LIN {X 0,Y 111.802,Z 888.457,A -85,B 0,C 180,E1 -29685.438,E2 -29685.438} C_VEL
LIN {X 0,Y 122.425,Z 878.603,A -85,B 0,C 180,E1 -29687.397,E2 -29687.397} C_VEL
LIN {X 0,Y 131.68,Z 868.339,A -85,B 0,C 180,E1 -29688.726,E2 -29688.726} C_VEL
LIN {X 0,Y 140.153,Z 857.045,A -85,B 0,C 180,E1 -29689.767,E2 -29689.767} C_VEL
LIN {X 0,Y 147.834,Z 844.571,A -85,B 0,C 180,E1 -29690.558,E2 -29690.558} C_VEL
LIN {X 0,Y 153.818,Z 832.536,A -85,B 0,C 180,E1 -29691.135,E2 -29691.135} C_VEL
LIN {X 0,Y 159.063,Z 819.023,A -85,B 0,C 180,E1 -29691.605,E2 -29691.605} C_VEL
LIN {X 0,Y 163.103,Z 804.721,A -85,B 0,C 180,E1 -29691.97,E2 -29691.97} C_VEL
LIN {X 0,Y 163.754,Z 801.83,A -85,B 0,C 180,E1 -29692.097,E2 -29692.097} C_VEL
LIN {X 0,Y 163.53,Z 800.148,A -85,B 0,C 180,E1 -29694.452,E2 -29694.452} C_VEL
LIN {X 0,Y 163.346,Z 799.523,A -85,B 0,C 180,E1 -29698.346,E2 -29698.346} C_VEL
LIN {X 0,Y 163.527,Z 800.407,A -85,B 0,C 180,E1 -29701.694,E2 -29701.694} C_VEL
LIN {X 0,Y 163.638,Z 801.813,A -85,B 0,C 180,E1 -29703.551,E2 -29703.551} C_VEL
LIN {X 0,Y 159.836,Z 815.926,A -85,B 0,C 180,E1 -29704.006,E2 -29704.006} C_VEL
LIN {X 0,Y 157.841,Z 821.597,A -85,B 0,C 180,E1 -29703.996,E2 -29703.996} C_VEL
LIN {X 0,Y 153.951,Z 830.589,A -85,B 0,C 180,E1 -29703.315,E2 -29703.315} C_VEL
LIN {X 0,Y 149.611,Z 839.251,A -85,B 0,C 180,E1 -29702.618,E2 -29702.618} C_VEL
LIN {X 0,Y 146.794,Z 844.327,A -85,B 0,C 180,E1 -29702.637,E2 -29702.637} C_VEL
LIN {X 0,Y 139.065,Z 856.566,A -85,B 0,C 180,E1 -29703.52,E2 -29703.52} C_VEL
LIN {X 0,Y 130.435,Z 867.719,A -85,B 0,C 180,E1 -29704.583,E2 -29704.583} C_VEL
LIN {X 0,Y 121.85,Z 877.024,A -85,B 0,C 180,E1 -29705.771,E2 -29705.771} C_VEL
LIN {X 0,Y 112.031,Z 885.993,A -85,B 0,C 180,E1 -29707.383,E2 -29707.383} C_VEL
LIN {X 0,Y 101.541,Z 894.03,A -85,B 0,C 180,E1 -29709.498,E2 -29709.498} C_VEL
LIN {X 0,Y 89.935,Z 901.363,A -85,B 0,C 180,E1 -29712.364,E2 -29712.364} C_VEL
LIN {X 0,Y 80.212,Z 906.465,A -85,B 0,C 180,E1 -29715.465,E2 -29715.465} C_VEL
LIN {X 0,Y 67.709,Z 911.76,A -85,B 0,C 180,E1 -29720.905,E2 -29720.905} C_VEL
LIN {X 0,Y 56.098,Z 915.48,A -85,B 0,C 180,E1 -29728.723,E2 -29728.723} C_VEL
LIN {X 0,Y 50.795,Z 916.801,A -85,B 0,C 180,E1 -29733.886,E2 -29733.886} C_VEL
LIN {X 0,Y 41.6,Z 918.426,A -85,B 0,C 180,E1 -29747.487,E2 -29747.487} C_VEL
LIN {X 0,Y 35.691,Z 918.717,A -85,B 0,C 180,E1 -29766.808,E2 -29766.808} C_VEL
LIN {X 0,Y 34.437,Z 918.369,A -85,B 0,C 180,E1 -29778.225,E2 -29778.225} C_VEL
LIN {X 0,Y 34.363,Z 917.697,A -85,B 0,C 180,E1 -29790.001,E2 -29790.001} C_VEL
LIN {X 0,Y 35.455,Z 916.701,A -85,B 0,C 180,E1 -29801.434,E2 -29801.434} C_VEL
LIN {X 0,Y 40.717,Z 913.712,A -85,B 0,C 180,E1 -29821.187,E2 -29821.187} C_VEL
LIN {X 0,Y 49.38,Z 909.289,A -85,B 0,C 180,E1 -29835.368,E2 -29835.368} C_VEL
LIN {X 0,Y 57.07,Z 904.914,A -85,B 0,C 180,E1 -29843.175,E2 -29843.175} C_VEL
LIN {X 0,Y 65.51,Z 899.589,A -85,B 0,C 180,E1 -29849.123,E2 -29849.123} C_VEL
LIN {X 0,Y 76.065,Z 891.943,A -85,B 0,C 180,E1 -29854.271,E2 -29854.271} C_VEL
LIN {X 0,Y 85.541,Z 883.95,A -85,B 0,C 180,E1 -29857.564,E2 -29857.564} C_VEL
LIN {X 0,Y 95.127,Z 874.337,A -85,B 0,C 180,E1 -29860.387,E2 -29860.387} C_VEL
LIN {X 0,Y 104.024,Z 863.685,A -85,B 0,C 180,E1 -29862.613,E2 -29862.613} C_VEL
LIN {X 0,Y 111.39,Z 853.168,A -85,B 0,C 180,E1 -29864.193,E2 -29864.193} C_VEL
LIN {X 0,Y 118.891,Z 840.267,A -85,B 0,C 180,E1 -29865.463,E2 -29865.463} C_VEL
LIN {X 0,Y 125.164,Z 826.62,A -85,B 0,C 180,E1 -29866.437,E2 -29866.437} C_VEL
LIN {X 0,Y 129.91,Z 812.825,A -85,B 0,C 180,E1 -29867.205,E2 -29867.205} C_VEL
LIN {X 0,Y 133.311,Z 798.837,A -85,B 0,C 180,E1 -29867.739,E2 -29867.739} C_VEL
LIN {X 0,Y 135.644,Z 782.896,A -85,B 0,C 180,E1 -29868.157,E2 -29868.157} C_VEL
LIN {X 0,Y 134.953,Z 780.303,A -85,B 0,C 180,E1 -29871.455,E2 -29871.455} C_VEL
LIN {X 0,Y 134.615,Z 777.995,A -85,B 0,C 180,E1 -29875.508,E2 -29875.508} C_VEL
LIN {X 0,Y 134.655,Z 777.956,A -85,B 0,C 180,E1 -29879.438,E2 -29879.438} C_VEL
LIN {X 0,Y 135.234,Z 781.24,A -85,B 0,C 180,E1 -29884.517,E2 -29884.517} C_VEL
LIN {X 0,Y 135.691,Z 783.05,A -85,B 0,C 180,E1 -29886.509,E2 -29886.509} C_VEL
LIN {X 0,Y 133.209,Z 800.155,A -85,B 0,C 180,E1 -29886.848,E2 -29886.848} C_VEL
LIN {X 0,Y 129.7,Z 814.546,A -85,B 0,C 180,E1 -29887.297,E2 -29887.297} C_VEL
LIN {X 0,Y 125.033,Z 827.951,A -85,B 0,C 180,E1 -29887.824,E2 -29887.824} C_VEL
LIN {X 0,Y 119.072,Z 841.078,A -85,B 0,C 180,E1 -29888.642,E2 -29888.642} C_VEL
LIN {X 0,Y 112.274,Z 853.019,A -85,B 0,C 180,E1 -29889.631,E2 -29889.631} C_VEL
LIN {X 0,Y 103.839,Z 865.127,A -85,B 0,C 180,E1 -29891.07,E2 -29891.07} C_VEL
LIN {X 0,Y 94.875,Z 875.902,A -85,B 0,C 180,E1 -29893.105,E2 -29893.105} C_VEL
LIN {X 0,Y 85.706,Z 885.152,A -85,B 0,C 180,E1 -29895.523,E2 -29895.523} C_VEL
LIN {X 0,Y 76.058,Z 893.431,A -85,B 0,C 180,E1 -29898.711,E2 -29898.711} C_VEL
LIN {X 0,Y 65.282,Z 901.369,A -85,B 0,C 180,E1 -29903.781,E2 -29903.781} C_VEL
LIN {X 0,Y 54.594,Z 908.033,A -85,B 0,C 180,E1 -29910.99,E2 -29910.99} C_VEL
LIN {X 0,Y 46.21,Z 912.763,A -85,B 0,C 180,E1 -29920.495,E2 -29920.495} C_VEL
LIN {X 0,Y 38.319,Z 917.014,A -85,B 0,C 180,E1 -29936.617,E2 -29936.617} C_VEL
LIN {X 0,Y 34.456,Z 919.808,A -85,B 0,C 180,E1 -29958.229,E2 -29958.229} C_VEL
LIN {X 0,Y 34.294,Z 920.676,A -85,B 0,C 180,E1 -29969.999,E2 -29969.999} C_VEL
LIN {X 0,Y 35.829,Z 921.312,A -85,B 0,C 180,E1 -29993.097,E2 -29993.097} C_VEL
LIN {X 0,Y 41.961,Z 920.62,A -85,B 0,C 180,E1 -30012.063,E2 -30012.063} C_VEL
LIN {X 0,Y 51.381,Z 918.607,A -85,B 0,C 180,E1 -30025.153,E2 -30025.153} C_VEL
LIN {X 0,Y 62.567,Z 915.214,A -85,B 0,C 180,E1 -30033.976,E2 -30033.976} C_VEL
LIN {X 0,Y 74.772,Z 910.35,A -85,B 0,C 180,E1 -30040.038,E2 -30040.038} C_VEL
LIN {X 0,Y 84.362,Z 905.692,A -85,B 0,C 180,E1 -30043.342,E2 -30043.342} C_VEL
LIN {X 0,Y 95.88,Z 898.946,A -85,B 0,C 180,E1 -30046.22,E2 -30046.22} C_VEL
LIN {X 0,Y 105.887,Z 891.893,A -85,B 0,C 180,E1 -30048.234,E2 -30048.234} C_VEL
LIN {X 0,Y 115.979,Z 883.447,A -85,B 0,C 180,E1 -30049.966,E2 -30049.966} C_VEL
LIN {X 0,Y 126.2,Z 873.292,A -85,B 0,C 180,E1 -30051.297,E2 -30051.297} C_VEL
LIN {X 0,Y 135.633,Z 861.932,A -85,B 0,C 180,E1 -30052.3,E2 -30052.3} C_VEL
LIN {X 0,Y 143.383,Z 850.655,A -85,B 0,C 180,E1 -30053.009,E2 -30053.009} C_VEL
LIN {X 0,Y 150.281,Z 838.353,A -85,B 0,C 180,E1 -30053.6,E2 -30053.6} C_VEL
LIN {X 0,Y 155.925,Z 825.739,A -85,B 0,C 180,E1 -30053.999,E2 -30053.999} C_VEL
LIN {X 0,Y 160.82,Z 811.209,A -85,B 0,C 180,E1 -30054.348,E2 -30054.348} C_VEL
LIN {X 0,Y 161.915,Z 807.143,A -85,B 0,C 180,E1 -30054.481,E2 -30054.481} C_VEL
LIN {X 0,Y 161.771,Z 806.425,A -85,B 0,C 180,E1 -30057.728,E2 -30057.728} C_VEL
LIN {X 0,Y 161.841,Z 807.145,A -85,B 0,C 180,E1 -30061.181,E2 -30061.181} C_VEL
LIN {X 0,Y 157.416,Z 821.391,A -85,B 0,C 180,E1 -30061.653,E2 -30061.653} C_VEL
LIN {X 0,Y 152.085,Z 834.135,A -85,B 0,C 180,E1 -30062.129,E2 -30062.129} C_VEL
LIN {X 0,Y 146.794,Z 844.327,A -85,B 0,C 180,E1 -30062.637,E2 -30062.637} C_VEL
LIN {X 0,Y 143.795,Z 849.42,A -85,B 0,C 180,E1 -30062.698,E2 -30062.698} C_VEL
LIN {X 0,Y 138.232,Z 857.51,A -85,B 0,C 180,E1 -30062.115,E2 -30062.115} C_VEL
LIN {X 0,Y 132.132,Z 865.2,A -85,B 0,C 180,E1 -30061.517,E2 -30061.517} C_VEL
LIN {X 0,Y 128.266,Z 869.655,A -85,B 0,C 180,E1 -30061.615,E2 -30061.615} C_VEL
LIN {X 0,Y 117.862,Z 880.277,A -85,B 0,C 180,E1 -30062.822,E2 -30062.822} C_VEL
LIN {X 0,Y 107.152,Z 889.318,A -85,B 0,C 180,E1 -30064.369,E2 -30064.369} C_VEL
LIN {X 0,Y 95.473,Z 897.454,A -85,B 0,C 180,E1 -30066.403,E2 -30066.403} C_VEL
LIN {X 0,Y 85.295,Z 903.281,A -85,B 0,C 180,E1 -30068.604,E2 -30068.604} C_VEL
LIN {X 0,Y 71.99,Z 909.482,A -85,B 0,C 180,E1 -30072.516,E2 -30072.516} C_VEL
LIN {X 0,Y 59.145,Z 914.001,A -85,B 0,C 180,E1 -30078.085,E2 -30078.085} C_VEL
LIN {X 0,Y 47.167,Z 917.027,A -85,B 0,C 180,E1 -30086.619,E2 -30086.619} C_VEL
LIN {X 0,Y 36.628,Z 918.681,A -85,B 0,C 180,E1 -30099.872,E2 -30099.872} C_VEL
LIN {X 0,Y 29.257,Z 918.999,A -85,B 0,C 180,E1 -30121.288,E2 -30121.288} C_VEL
LIN {X 0,Y 27.252,Z 918.006,A -85,B 0,C 180,E1 -30150.001,E2 -30150.001} C_VEL
LIN {X 0,Y 28.537,Z 917.023,A -85,B 0,C 180,E1 -30164.259,E2 -30164.259} C_VEL
LIN {X 0,Y 34.867,Z 914.062,A -85,B 0,C 180,E1 -30187.209,E2 -30187.209} C_VEL
LIN {X 0,Y 44.696,Z 909.67,A -85,B 0,C 180,E1 -30201.834,E2 -30201.834} C_VEL
LIN {X 0,Y 53.135,Z 905.327,A -85,B 0,C 180,E1 -30209.289,E2 -30209.289} C_VEL
LIN {X 0,Y 63.735,Z 899.04,A -85,B 0,C 180,E1 -30215.468,E2 -30215.468} C_VEL
LIN {X 0,Y 73.277,Z 892.43,A -85,B 0,C 180,E1 -30219.249,E2 -30219.249} C_VEL
LIN {X 0,Y 83.101,Z 884.483,A -85,B 0,C 180,E1 -30222.072,E2 -30222.072} C_VEL
LIN {X 0,Y 92.995,Z 874.921,A -85,B 0,C 180,E1 -30224.489,E2 -30224.489} C_VEL
LIN {X 0,Y 102.141,Z 864.331,A -85,B 0,C 180,E1 -30226.388,E2 -30226.388} C_VEL
LIN {X 0,Y 109.679,Z 853.893,A -85,B 0,C 180,E1 -30227.74,E2 -30227.74} C_VEL
LIN {X 0,Y 117.318,Z 841.095,A -85,B 0,C 180,E1 -30228.803,E2 -30228.803} C_VEL
LIN {X 0,Y 123.229,Z 828.693,A -85,B 0,C 180,E1 -30229.546,E2 -30229.546} C_VEL
LIN {X 0,Y 128.36,Z 814.653,A -85,B 0,C 180,E1 -30230.247,E2 -30230.247} C_VEL
LIN {X 0,Y 132.029,Z 800.539,A -85,B 0,C 180,E1 -30230.714,E2 -30230.714} C_VEL
LIN {X 0,Y 134.104,Z 787.89,A -85,B 0,C 180,E1 -30231.065,E2 -30231.065} C_VEL
LIN {X 0,Y 133.724,Z 784.916,A -85,B 0,C 180,E1 -30236.232,E2 -30236.232} C_VEL
LIN {X 0,Y 133.754,Z 785.03,A -85,B 0,C 180,E1 -30239.058,E2 -30239.058} C_VEL
LIN {X 0,Y 134.15,Z 787.871,A -85,B 0,C 180,E1 -30243.573,E2 -30243.573} C_VEL
LIN {X 0,Y 131.673,Z 802.747,A -85,B 0,C 180,E1 -30243.89,E2 -30243.89} C_VEL
LIN {X 0,Y 127.815,Z 817.044,A -85,B 0,C 180,E1 -30244.282,E2 -30244.282} C_VEL
LIN {X 0,Y 122.968,Z 830.024,A -85,B 0,C 180,E1 -30244.714,E2 -30244.714} C_VEL
LIN {X 0,Y 116.48,Z 843.438,A -85,B 0,C 180,E1 -30245.401,E2 -30245.401} C_VEL
LIN {X 0,Y 108.718,Z 856.198,A -85,B 0,C 180,E1 -30246.324,E2 -30246.324} C_VEL
LIN {X 0,Y 100.137,Z 867.714,A -85,B 0,C 180,E1 -30247.538,E2 -30247.538} C_VEL
LIN {X 0,Y 90.826,Z 878.182,A -85,B 0,C 180,E1 -30249.394,E2 -30249.394} C_VEL
LIN {X 0,Y 80.726,Z 887.602,A -85,B 0,C 180,E1 -30251.638,E2 -30251.638} C_VEL
LIN {X 0,Y 70.786,Z 895.429,A -85,B 0,C 180,E1 -30254.523,E2 -30254.523} C_VEL
LIN {X 0,Y 59.577,Z 902.928,A -85,B 0,C 180,E1 -30259.311,E2 -30259.311} C_VEL
LIN {X 0,Y 47.421,Z 909.647,A -85,B 0,C 180,E1 -30267.221,E2 -30267.221} C_VEL
LIN {X 0,Y 36.902,Z 914.711,A -85,B 0,C 180,E1 -30280.374,E2 -30280.374} C_VEL
LIN {X 0,Y 29.369,Z 918.251,A -85,B 0,C 180,E1 -30301.405,E2 -30301.405} C_VEL
LIN {X 0,Y 27.512,Z 919.485,A -85,B 0,C 180,E1 -30315.198,E2 -30315.198} C_VEL
LIN {X 0,Y 27.203,Z 920.369,A -85,B 0,C 180,E1 -30329.999,E2 -30329.999} C_VEL
LIN {X 0,Y 29.399,Z 921.031,A -85,B 0,C 180,E1 -30358.56,E2 -30358.56} C_VEL
LIN {X 0,Y 36.974,Z 920.369,A -85,B 0,C 180,E1 -30379.49,E2 -30379.49} C_VEL
LIN {X 0,Y 47.66,Z 918.39,A -85,B 0,C 180,E1 -30392.221,E2 -30392.221} C_VEL
LIN {X 0,Y 59.779,Z 915.031,A -85,B 0,C 180,E1 -30400.139,E2 -30400.139} C_VEL
LIN {X 0,Y 72.643,Z 910.198,A -85,B 0,C 180,E1 -30405.344,E2 -30405.344} C_VEL
LIN {X 0,Y 82.598,Z 905.563,A -85,B 0,C 180,E1 -30408.094,E2 -30408.094} C_VEL
LIN {X 0,Y 94.434,Z 898.857,A -85,B 0,C 180,E1 -30410.434,E2 -30410.434} C_VEL
LIN {X 0,Y 106.377,Z 890.533,A -85,B 0,C 180,E1 -30412.308,E2 -30412.308} C_VEL
LIN {X 0,Y 116.677,Z 881.879,A -85,B 0,C 180,E1 -30413.652,E2 -30413.652} C_VEL
LIN {X 0,Y 127.053,Z 871.412,A -85,B 0,C 180,E1 -30414.67,E2 -30414.67} C_VEL
LIN {X 0,Y 135.733,Z 860.891,A -85,B 0,C 180,E1 -30415.36,E2 -30415.36} C_VEL
LIN {X 0,Y 143.564,Z 849.45,A -85,B 0,C 180,E1 -30415.892,E2 -30415.892} C_VEL
LIN {X 0,Y 150.532,Z 836.923,A -85,B 0,C 180,E1 -30416.332,E2 -30416.332} C_VEL
LIN {X 0,Y 156.136,Z 824.202,A -85,B 0,C 180,E1 -30416.634,E2 -30416.634} C_VEL
LIN {X 0,Y 159.878,Z 813.372,A -85,B 0,C 180,E1 -30416.868,E2 -30416.868} C_VEL
LIN {X 0,Y 159.853,Z 813.351,A -85,B 0,C 180,E1 -30418.793,E2 -30418.793} C_VEL
LIN {X 0,Y 155.255,Z 826.323,A -85,B 0,C 180,E1 -30419.227,E2 -30419.227} C_VEL
LIN {X 0,Y 149.348,Z 839.106,A -85,B 0,C 180,E1 -30419.621,E2 -30419.621} C_VEL
LIN {X 0,Y 141.764,Z 852.028,A -85,B 0,C 180,E1 -30420.274,E2 -30420.274} C_VEL
LIN {X 0,Y 133.555,Z 863.379,A -85,B 0,C 180,E1 -30421.067,E2 -30421.067} C_VEL
LIN {X 0,Y 128.266,Z 869.655,A -85,B 0,C 180,E1 -30421.615,E2 -30421.615} C_VEL
LIN {X 0,Y 124.238,Z 874.015,A -85,B 0,C 180,E1 -30421.73,E2 -30421.73} C_VEL
LIN {X 0,Y 117.171,Z 880.865,A -85,B 0,C 180,E1 -30421.118,E2 -30421.118} C_VEL
LIN {X 0,Y 109.693,Z 887.223,A -85,B 0,C 180,E1 -30420.52,E2 -30420.52} C_VEL
LIN {X 0,Y 105.003,Z 890.749,A -85,B 0,C 180,E1 -30420.76,E2 -30420.76} C_VEL
LIN {X 0,Y 93.199,Z 898.593,A -85,B 0,C 180,E1 -30422.35,E2 -30422.35} C_VEL
LIN {X 0,Y 81.065,Z 905.127,A -85,B 0,C 180,E1 -30424.44,E2 -30424.44} C_VEL
LIN {X 0,Y 67.385,Z 910.895,A -85,B 0,C 180,E1 -30427.773,E2 -30427.773} C_VEL
LIN {X 0,Y 57.319,Z 914.199,A -85,B 0,C 180,E1 -30431.22,E2 -30431.22} C_VEL
LIN {X 0,Y 43.9,Z 917.344,A -85,B 0,C 180,E1 -30438.677,E2 -30438.677} C_VEL
LIN {X 0,Y 32.498,Z 918.936,A -85,B 0,C 180,E1 -30450.116,E2 -30450.116} C_VEL
LIN {X 0,Y 23.219,Z 919.283,A -85,B 0,C 180,E1 -30472.746,E2 -30472.746} C_VEL
LIN {X 0,Y 20.655,Z 918.961,A -85,B 0,C 180,E1 -30490.11,E2 -30490.11} C_VEL
LIN {X 0,Y 20.124,Z 918.316,A -85,B 0,C 180,E1 -30510.002,E2 -30510.002} C_VEL
LIN {X 0,Y 21.723,Z 917.346,A -85,B 0,C 180,E1 -30528.878,E2 -30528.878} C_VEL
LIN {X 0,Y 29.537,Z 914.413,A -85,B 0,C 180,E1 -30555.549,E2 -30555.549} C_VEL
LIN {X 0,Y 40.698,Z 910.052,A -85,B 0,C 180,E1 -30569.706,E2 -30569.706} C_VEL
LIN {X 0,Y 53.054,Z 904.133,A -85,B 0,C 180,E1 -30578.018,E2 -30578.018} C_VEL
LIN {X 0,Y 64.417,Z 897.464,A -85,B 0,C 180,E1 -30582.68,E2 -30582.68} C_VEL
LIN {X 0,Y 76.142,Z 889.145,A -85,B 0,C 180,E1 -30585.738,E2 -30585.738} C_VEL
LIN {X 0,Y 86.28,Z 880.485,A -85,B 0,C 180,E1 -30587.816,E2 -30587.816} C_VEL
LIN {X 0,Y 96.446,Z 870.016,A -85,B 0,C 180,E1 -30589.657,E2 -30589.657} C_VEL
LIN {X 0,Y 104.971,Z 859.456,A -85,B 0,C 180,E1 -30590.949,E2 -30590.949} C_VEL
LIN {X 0,Y 112.714,Z 847.905,A -85,B 0,C 180,E1 -30591.831,E2 -30591.831} C_VEL
LIN {X 0,Y 119.611,Z 835.209,A -85,B 0,C 180,E1 -30592.538,E2 -30592.538} C_VEL
LIN {X 0,Y 125.291,Z 821.849,A -85,B 0,C 180,E1 -30593.132,E2 -30593.132} C_VEL
LIN {X 0,Y 129.746,Z 807.713,A -85,B 0,C 180,E1 -30593.629,E2 -30593.629} C_VEL
LIN {X 0,Y 132.743,Z 793.388,A -85,B 0,C 180,E1 -30594.016,E2 -30594.016} C_VEL
LIN {X 0,Y 132.766,Z 791.859,A -85,B 0,C 180,E1 -30596.965,E2 -30596.965} C_VEL
LIN {X 0,Y 132.78,Z 792.026,A -85,B 0,C 180,E1 -30598.625,E2 -30598.625} C_VEL
LIN {X 0,Y 132.804,Z 793.19,A -85,B 0,C 180,E1 -30600.621,E2 -30600.621} C_VEL
LIN {X 0,Y 129.73,Z 808.132,A -85,B 0,C 180,E1 -30600.906,E2 -30600.906} C_VEL
LIN {X 0,Y 125.215,Z 822.442,A -85,B 0,C 180,E1 -30601.212,E2 -30601.212} C_VEL
LIN {X 0,Y 119.524,Z 835.81,A -85,B 0,C 180,E1 -30601.601,E2 -30601.601} C_VEL
LIN {X 0,Y 112.53,Z 848.682,A -85,B 0,C 180,E1 -30602.168,E2 -30602.168} C_VEL
LIN {X 0,Y 104.676,Z 860.379,A -85,B 0,C 180,E1 -30602.889,E2 -30602.889} C_VEL
LIN {X 0,Y 96.792,Z 870.187,A -85,B 0,C 180,E1 -30603.819,E2 -30603.819} C_VEL
LIN {X 0,Y 86.478,Z 880.927,A -85,B 0,C 180,E1 -30605.401,E2 -30605.401} C_VEL
LIN {X 0,Y 76.163,Z 889.83,A -85,B 0,C 180,E1 -30607.265,E2 -30607.265} C_VEL
LIN {X 0,Y 65.959,Z 897.236,A -85,B 0,C 180,E1 -30609.732,E2 -30609.732} C_VEL
LIN {X 0,Y 54.301,Z 904.329,A -85,B 0,C 180,E1 -30613.898,E2 -30613.898} C_VEL
LIN {X 0,Y 44.592,Z 909.246,A -85,B 0,C 180,E1 -30618.976,E2 -30618.976} C_VEL
LIN {X 0,Y 32.728,Z 914.344,A -85,B 0,C 180,E1 -30630.798,E2 -30630.798} C_VEL
LIN {X 0,Y 23.344,Z 917.913,A -85,B 0,C 180,E1 -30652.976,E2 -30652.976} C_VEL
LIN {X 0,Y 20.082,Z 920.06,A -85,B 0,C 180,E1 -30689.998,E2 -30689.998} C_VEL
LIN {X 0,Y 23.389,Z 920.75,A -85,B 0,C 180,E1 -30726.938,E2 -30726.938} C_VEL
LIN {X 0,Y 32.793,Z 920.116,A -85,B 0,C 180,E1 -30749.006,E2 -30749.006} C_VEL
LIN {X 0,Y 44.779,Z 918.169,A -85,B 0,C 180,E1 -30760.336,E2 -30760.336} C_VEL
LIN {X 0,Y 57.743,Z 914.848,A -85,B 0,C 180,E1 -30766.827,E2 -30766.827} C_VEL
LIN {X 0,Y 71.173,Z 910.047,A -85,B 0,C 180,E1 -30770.909,E2 -30770.909} C_VEL
LIN {X 0,Y 81.426,Z 905.43,A -85,B 0,C 180,E1 -30773.014,E2 -30773.014} C_VEL
LIN {X 0,Y 93.512,Z 898.763,A -85,B 0,C 180,E1 -30774.755,E2 -30774.755} C_VEL
LIN {X 0,Y 105.659,Z 890.493,A -85,B 0,C 180,E1 -30776.139,E2 -30776.139} C_VEL
LIN {X 0,Y 116.106,Z 881.886,A -85,B 0,C 180,E1 -30777.145,E2 -30777.145} C_VEL
LIN {X 0,Y 126.591,Z 871.475,A -85,B 0,C 180,E1 -30777.866,E2 -30777.866} C_VEL
LIN {X 0,Y 126.544,Z 871.488,A -85,B 0,C 180,E1 -30778.553,E2 -30778.553} C_VEL
LIN {X 0,Y 115.966,Z 881.891,A -85,B 0,C 180,E1 -30779.514,E2 -30779.514} C_VEL
LIN {X 0,Y 105.003,Z 890.749,A -85,B 0,C 180,E1 -30780.76,E2 -30780.76} C_VEL
LIN {X 0,Y 99.654,Z 894.512,A -85,B 0,C 180,E1 -30781.1,E2 -30781.1} C_VEL
LIN {X 0,Y 90.388,Z 900.206,A -85,B 0,C 180,E1 -30780.548,E2 -30780.548} C_VEL
LIN {X 0,Y 82.721,Z 904.33,A -85,B 0,C 180,E1 -30779.918,E2 -30779.918} C_VEL
LIN {X 0,Y 76.815,Z 907.092,A -85,B 0,C 180,E1 -30779.978,E2 -30779.978} C_VEL
LIN {X 0,Y 74.835,Z 907.933,A -85,B 0,C 180,E1 -30780.213,E2 -30780.213} C_VEL
LIN {X 0,Y 63.304,Z 912.291,A -85,B 0,C 180,E1 -30782.332,E2 -30782.332} C_VEL
LIN {X 0,Y 49.486,Z 916.117,A -85,B 0,C 180,E1 -30786.212,E2 -30786.212} C_VEL
LIN {X 0,Y 36.032,Z 918.504,A -85,B 0,C 180,E1 -30792.778,E2 -30792.778} C_VEL
LIN {X 0,Y 23.427,Z 919.545,A -85,B 0,C 180,E1 -30805.849,E2 -30805.849} C_VEL
LIN {X 0,Y 14.153,Z 919.257,A -85,B 0,C 180,E1 -30840.229,E2 -30840.229} C_VEL
LIN {X 0,Y 12.997,Z 918.625,A -85,B 0,C 180,E1 -30870.003,E2 -30870.003} C_VEL
LIN {X 0,Y 15.197,Z 917.668,A -85,B 0,C 180,E1 -30897.549,E2 -30897.549} C_VEL
LIN {X 0,Y 25.102,Z 914.763,A -85,B 0,C 180,E1 -30927.137,E2 -30927.137} C_VEL
LIN {X 0,Y 37.63,Z 910.433,A -85,B 0,C 180,E1 -30939.043,E2 -30939.043} C_VEL
LIN {X 0,Y 50.828,Z 904.557,A -85,B 0,C 180,E1 -30945.444,E2 -30945.444} C_VEL
LIN {X 0,Y 62.677,Z 897.929,A -85,B 0,C 180,E1 -30948.86,E2 -30948.86} C_VEL
LIN {X 0,Y 74.716,Z 889.655,A -85,B 0,C 180,E1 -30950.996,E2 -30950.996} C_VEL
LIN {X 0,Y 85.07,Z 881.042,A -85,B 0,C 180,E1 -30952.471,E2 -30952.471} C_VEL
LIN {X 0,Y 95.432,Z 870.629,A -85,B 0,C 180,E1 -30953.827,E2 -30953.827} C_VEL
LIN {X 0,Y 104.095,Z 860.139,A -85,B 0,C 180,E1 -30954.784,E2 -30954.784} C_VEL
LIN {X 0,Y 111.931,Z 848.676,A -85,B 0,C 180,E1 -30955.403,E2 -30955.403} C_VEL
LIN {X 0,Y 118.901,Z 836.101,A -85,B 0,C 180,E1 -30955.915,E2 -30955.915} C_VEL
LIN {X 0,Y 124.381,Z 823.592,A -85,B 0,C 180,E1 -30956.334,E2 -30956.334} C_VEL
LIN {X 0,Y 129.008,Z 809.581,A -85,B 0,C 180,E1 -30956.725,E2 -30956.725} C_VEL
LIN {X 0,Y 131.489,Z 799.151,A -85,B 0,C 180,E1 -30956.935,E2 -30956.935} C_VEL
LIN {X 0,Y 131.547,Z 798.848,A -85,B 0,C 180,E1 -30957.144,E2 -30957.144} C_VEL
LIN {X 0,Y 131.554,Z 798.839,A -85,B 0,C 180,E1 -30957.627,E2 -30957.627} C_VEL
LIN {X 0,Y 128.021,Z 813.059,A -85,B 0,C 180,E1 -30957.833,E2 -30957.833} C_VEL
LIN {X 0,Y 123.033,Z 827.133,A -85,B 0,C 180,E1 -30958.033,E2 -30958.033} C_VEL
LIN {X 0,Y 116.89,Z 840.204,A -85,B 0,C 180,E1 -30958.342,E2 -30958.342} C_VEL
LIN {X 0,Y 109.843,Z 852.15,A -85,B 0,C 180,E1 -30958.671,E2 -30958.671} C_VEL
LIN {X 0,Y 101.038,Z 864.266,A -85,B 0,C 180,E1 -30959.211,E2 -30959.211} C_VEL
LIN {X 0,Y 92.511,Z 874.036,A -85,B 0,C 180,E1 -30959.999,E2 -30959.999} C_VEL
LIN {X 0,Y 82.592,Z 883.548,A -85,B 0,C 180,E1 -30960.985,E2 -30960.985} C_VEL
LIN {X 0,Y 72.097,Z 891.965,A -85,B 0,C 180,E1 -30962.327,E2 -30962.327} C_VEL
LIN {X 0,Y 59.931,Z 900.014,A -85,B 0,C 180,E1 -30964.584,E2 -30964.584} C_VEL
LIN {X 0,Y 49.609,Z 905.677,A -85,B 0,C 180,E1 -30967.393,E2 -30967.393} C_VEL
LIN {X 0,Y 39.456,Z 910.296,A -85,B 0,C 180,E1 -30971.567,E2 -30971.567} C_VEL
LIN {X 0,Y 29.7,Z 913.976,A -85,B 0,C 180,E1 -30978.817,E2 -30978.817} C_VEL
LIN {X 0,Y 18.144,Z 917.574,A -85,B 0,C 180,E1 -30999.22,E2 -30999.22} C_VEL
LIN {X 0,Y 14.191,Z 918.838,A -85,B 0,C 180,E1 -31020.31,E2 -31020.31} C_VEL
LIN {X 0,Y 12.968,Z 919.752,A -85,B 0,C 180,E1 -31049.997,E2 -31049.997} C_VEL
LIN {X 0,Y 18.196,Z 920.468,A -85,B 0,C 180,E1 -31100.575,E2 -31100.575} C_VEL
LIN {X 0,Y 29.757,Z 919.862,A -85,B 0,C 180,E1 -31120.857,E2 -31120.857} C_VEL
LIN {X 0,Y 42.902,Z 917.944,A -85,B 0,C 180,E1 -31129.382,E2 -31129.382} C_VEL
LIN {X 0,Y 56.541,Z 914.66,A -85,B 0,C 180,E1 -31133.921,E2 -31133.921} C_VEL
LIN {X 0,Y 70.4,Z 909.895,A -85,B 0,C 180,E1 -31136.649,E2 -31136.649} C_VEL
LIN {X 0,Y 80.869,Z 905.294,A -85,B 0,C 180,E1 -31138.034,E2 -31138.034} C_VEL
LIN {X 0,Y 84.369,Z 903.524,A -85,B 0,C 180,E1 -31138.387,E2 -31138.387} C_VEL
LIN {X 0,Y 84.351,Z 903.511,A -85,B 0,C 180,E1 -31138.911,E2 -31138.911} C_VEL
LIN {X 0,Y 74.835,Z 907.933,A -85,B 0,C 180,E1 -31140.213,E2 -31140.213} C_VEL
LIN {X 0,Y 67.077,Z 910.991,A -85,B 0,C 180,E1 -31140.996,E2 -31140.996} C_VEL
LIN {X 0,Y 59.107,Z 913.613,A -85,B 0,C 180,E1 -31141.122,E2 -31141.122} C_VEL
LIN {X 0,Y 48.273,Z 916.457,A -85,B 0,C 180,E1 -31140.785,E2 -31140.785} C_VEL
LIN {X 0,Y 37.279,Z 918.46,A -85,B 0,C 180,E1 -31141.124,E2 -31141.124} C_VEL
LIN {X 0,Y 31.799,Z 919.08,A -85,B 0,C 180,E1 -31142.463,E2 -31142.463} C_VEL
LIN {X 0,Y 21.302,Z 919.814,A -85,B 0,C 180,E1 -31148.207,E2 -31148.207} C_VEL
LIN {X 0,Y 8.697,Z 919.554,A -85,B 0,C 180,E1 -31176.095,E2 -31176.095} C_VEL
LIN {X 0,Y 5.887,Z 918.934,A -85,B 0,C 180,E1 -31230.007,E2 -31230.007} C_VEL
LIN {X 0,Y 9.493,Z 917.99,A -85,B 0,C 180,E1 -31277.763,E2 -31277.763} C_VEL
LIN {X 0,Y 22.073,Z 915.114,A -85,B 0,C 180,E1 -31302.793,E2 -31302.793} C_VEL
LIN {X 0,Y 35.715,Z 910.815,A -85,B 0,C 180,E1 -31309.716,E2 -31309.716} C_VEL
LIN {X 0,Y 49.526,Z 904.975,A -85,B 0,C 180,E1 -31313.39,E2 -31313.39} C_VEL
LIN {X 0,Y 61.703,Z 898.387,A -85,B 0,C 180,E1 -31315.309,E2 -31315.309} C_VEL
LIN {X 0,Y 70.441,Z 892.668,A -85,B 0,C 180,E1 -31316.139,E2 -31316.139} C_VEL
LIN {X 0,Y 70.394,Z 892.719,A -85,B 0,C 180,E1 -31316.746,E2 -31316.746} C_VEL
LIN {X 0,Y 58.019,Z 900.586,A -85,B 0,C 180,E1 -31317.942,E2 -31317.942} C_VEL
LIN {X 0,Y 45.68,Z 906.897,A -85,B 0,C 180,E1 -31319.618,E2 -31319.618} C_VEL
LIN {X 0,Y 31.682,Z 912.491,A -85,B 0,C 180,E1 -31323.377,E2 -31323.377} C_VEL
LIN {X 0,Y 21.35,Z 915.602,A -85,B 0,C 180,E1 -31329.038,E2 -31329.038} C_VEL
LIN {X 0,Y 8.73,Z 918.514,A -85,B 0,C 180,E1 -31356.38,E2 -31356.38} C_VEL
LIN {X 0,Y 5.868,Z 919.444,A -85,B 0,C 180,E1 -31409.993,E2 -31409.993} C_VEL
LIN {X 0,Y 14.728,Z 920.186,A -85,B 0,C 180,E1 -31482.618,E2 -31482.618} C_VEL
LIN {X 0,Y 28.231,Z 919.608,A -85,B 0,C 180,E1 -31494.713,E2 -31494.713} C_VEL
LIN {X 0,Y 42.174,Z 917.717,A -85,B 0,C 180,E1 -31498.993,E2 -31498.993} C_VEL
LIN {X 0,Y 42.17,Z 917.708,A -85,B 0,C 180,E1 -31499.37,E2 -31499.37} C_VEL
LIN {X 0,Y 31.799,Z 919.08,A -85,B 0,C 180,E1 -31502.463,E2 -31502.463} C_VEL
LIN {X 0,Y 31.799,Z 919.08,A -85,B 0,C 180,E1 -31502.463,E2 -31502.463}

QRS_NEXT_CUT()

QRS_NEXT()
QRS_HOME()

END
